LIN {X 0,Y 571.544,Z 581.049,A -85,B 0,C 180,E1 -1504.136,E2 -1504.136} C_VEL
LIN {X 0,Y 571.308,Z 601.407,A -85,B 0,C 180,E1 -1504.632,E2 -1504.632} C_VEL
LIN {X 0,Y 570.995,Z 621.202,A -85,B 0,C 180,E1 -1505.305,E2 -1505.305} C_VEL
LIN {X 0,Y 570.609,Z 639.891,A -85,B 0,C 180,E1 -1506.125,E2 -1506.125} C_VEL
LIN {X 0,Y 570.21,Z 658.766,A -85,B 0,C 180,E1 -1507.147,E2 -1507.147} C_VEL
LIN {X 0,Y 569.785,Z 677.478,A -85,B 0,C 180,E1 -1508.378,E2 -1508.378} C_VEL
LIN {X 0,Y 569.391,Z 694.356,A -85,B 0,C 180,E1 -1509.704,E2 -1509.704} C_VEL
LIN {X 0,Y 569.023,Z 710.417,A -85,B 0,C 180,E1 -1511.191,E2 -1511.191} C_VEL
LIN {X 0,Y 568.698,Z 725.365,A -85,B 0,C 180,E1 -1512.822,E2 -1512.822} C_VEL
LIN {X 0,Y 568.433,Z 739.137,A -85,B 0,C 180,E1 -1514.598,E2 -1514.598} C_VEL
LIN {X 0,Y 568.219,Z 751.298,A -85,B 0,C 180,E1 -1516.467,E2 -1516.467} C_VEL
LIN {X 0,Y 568.077,Z 761.373,A -85,B 0,C 180,E1 -1518.323,E2 -1518.323} C_VEL
LIN {X 0,Y 567.993,Z 770.289,A -85,B 0,C 180,E1 -1520.328,E2 -1520.328} C_VEL
LIN {X 0,Y 567.945,Z 777.475,A -85,B 0,C 180,E1 -1522.372,E2 -1522.372} C_VEL
LIN {X 0,Y 567.92,Z 782.732,A -85,B 0,C 180,E1 -1524.343,E2 -1524.343} C_VEL
LIN {X 0,Y 567.908,Z 786.402,A -85,B 0,C 180,E1 -1526.367,E2 -1526.367} C_VEL
LIN {X 0,Y 567.902,Z 788.441,A -85,B 0,C 180,E1 -1528.387,E2 -1528.387} C_VEL
LIN {X 0,Y 567.9,Z 788.895,A -85,B 0,C 180,E1 -1530.505,E2 -1530.505} C_VEL
LIN {X 0,Y 567.907,Z 787.727,A -85,B 0,C 180,E1 -1532.524,E2 -1532.524} C_VEL
LIN {X 0,Y 567.913,Z 784.97,A -85,B 0,C 180,E1 -1534.545,E2 -1534.545} C_VEL
LIN {X 0,Y 567.931,Z 780.48,A -85,B 0,C 180,E1 -1536.572,E2 -1536.572} C_VEL
LIN {X 0,Y 567.969,Z 774.262,A -85,B 0,C 180,E1 -1538.607,E2 -1538.607} C_VEL
LIN {X 0,Y 568.028,Z 766.175,A -85,B 0,C 180,E1 -1540.652,E2 -1540.652} C_VEL
LIN {X 0,Y 568.143,Z 756.561,A -85,B 0,C 180,E1 -1542.606,E2 -1542.606} C_VEL
LIN {X 0,Y 568.325,Z 745.488,A -85,B 0,C 180,E1 -1544.468,E2 -1544.468} C_VEL
LIN {X 0,Y 568.551,Z 732.933,A -85,B 0,C 180,E1 -1546.238,E2 -1546.238} C_VEL
LIN {X 0,Y 568.832,Z 718.879,A -85,B 0,C 180,E1 -1547.916,E2 -1547.916} C_VEL
LIN {X 0,Y 569.169,Z 703.833,A -85,B 0,C 180,E1 -1549.445,E2 -1549.445} C_VEL
LIN {X 0,Y 569.551,Z 687.283,A -85,B 0,C 180,E1 -1550.878,E2 -1550.878} C_VEL
LIN {X 0,Y 569.976,Z 668.941,A -85,B 0,C 180,E1 -1552.213,E2 -1552.213} C_VEL
LIN {X 0,Y 570.388,Z 650.263,A -85,B 0,C 180,E1 -1553.34,E2 -1553.34} C_VEL
LIN {X 0,Y 570.784,Z 631.791,A -85,B 0,C 180,E1 -1554.255,E2 -1554.255} C_VEL
LIN {X 0,Y 571.16,Z 611.854,A -85,B 0,C 180,E1 -1555.038,E2 -1555.038} C_VEL
LIN {X 0,Y 571.428,Z 591.582,A -85,B 0,C 180,E1 -1555.63,E2 -1555.63} C_VEL
LIN {X 0,Y 571.638,Z 571.154,A -85,B 0,C 180,E1 -1556.037,E2 -1556.037} C_VEL
LIN {X 0,Y 572.618,Z 333.536,A -85,B 0,C 180,E1 -1559.297,E2 -1559.297} C_VEL
LIN {X 0,Y 572.442,Z 320.457,A -85,B 0,C 180,E1 -1559.491,E2 -1559.491} C_VEL
LIN {X 0,Y 571.564,Z 314.836,A -85,B 0,C 180,E1 -1559.646,E2 -1559.646} C_VEL
LIN {X 0,Y 572.165,Z 276.654,A -85,B 0,C 180,E1 -1562.244,E2 -1562.244} C_VEL
LIN {X 0,Y 568.247,Z 266.023,A -85,B 0,C 180,E1 -1563.279,E2 -1563.279} C_VEL
LIN {X 0,Y 568.203,Z 265.709,A -85,B 0,C 180,E1 -1564.149,E2 -1564.149} C_VEL
LIN {X 0,Y 568.186,Z 265.71,A -85,B 0,C 180,E1 -1567.509,E2 -1567.509} C_VEL
LIN {X 0,Y 568.221,Z 265.707,A -85,B 0,C 180,E1 -1570.756,E2 -1570.756} C_VEL
LIN {X 0,Y 568.185,Z 265.706,A -85,B 0,C 180,E1 -1574.036,E2 -1574.036} C_VEL
LIN {X 0,Y 568.192,Z 265.71,A -85,B 0,C 180,E1 -1577.356,E2 -1577.356} C_VEL
LIN {X 0,Y 568.224,Z 265.704,A -85,B 0,C 180,E1 -1580.577,E2 -1580.577} C_VEL
LIN {X 0,Y 568.171,Z 265.709,A -85,B 0,C 180,E1 -1583.752,E2 -1583.752} C_VEL
LIN {X 0,Y 568.219,Z 265.709,A -85,B 0,C 180,E1 -1586.942,E2 -1586.942} C_VEL
LIN {X 0,Y 568.251,Z 265.927,A -85,B 0,C 180,E1 -1589.055,E2 -1589.055} C_VEL
LIN {X 0,Y 571.301,Z 275.947,A -85,B 0,C 180,E1 -1590.08,E2 -1590.08} C_VEL
LIN {X 0,Y 570.614,Z 317.064,A -85,B 0,C 180,E1 -1593.297,E2 -1593.297} C_VEL
LIN {X 0,Y 570.322,Z 342.297,A -85,B 0,C 180,E1 -1595.215,E2 -1595.215} C_VEL
LIN {X 0,Y 571.283,Z 349.569,A -85,B 0,C 180,E1 -1595.372,E2 -1595.372} C_VEL
LIN {X 0,Y 570.541,Z 559.942,A -85,B 0,C 180,E1 -1598.191,E2 -1598.191} C_VEL
LIN {X 0,Y 570.341,Z 579.649,A -85,B 0,C 180,E1 -1598.652,E2 -1598.652} C_VEL
LIN {X 0,Y 570.092,Z 598.197,A -85,B 0,C 180,E1 -1599.278,E2 -1599.278} C_VEL
LIN {X 0,Y 569.786,Z 616.477,A -85,B 0,C 180,E1 -1600.097,E2 -1600.097} C_VEL
LIN {X 0,Y 569.463,Z 634.177,A -85,B 0,C 180,E1 -1601.099,E2 -1601.099} C_VEL
LIN {X 0,Y 569.137,Z 650.753,A -85,B 0,C 180,E1 -1602.254,E2 -1602.254} C_VEL
LIN {X 0,Y 568.827,Z 666.254,A -85,B 0,C 180,E1 -1603.561,E2 -1603.561} C_VEL
LIN {X 0,Y 568.552,Z 680.636,A -85,B 0,C 180,E1 -1605.018,E2 -1605.018} C_VEL
LIN {X 0,Y 568.336,Z 693.477,A -85,B 0,C 180,E1 -1606.572,E2 -1606.572} C_VEL
LIN {X 0,Y 568.164,Z 704.809,A -85,B 0,C 180,E1 -1608.221,E2 -1608.221} C_VEL
LIN {X 0,Y 568.047,Z 714.647,A -85,B 0,C 180,E1 -1609.965,E2 -1609.965} C_VEL
LIN {X 0,Y 567.968,Z 722.967,A -85,B 0,C 180,E1 -1611.802,E2 -1611.802} C_VEL
LIN {X 0,Y 567.933,Z 729.712,A -85,B 0,C 180,E1 -1613.734,E2 -1613.734} C_VEL
LIN {X 0,Y 567.911,Z 734.541,A -85,B 0,C 180,E1 -1615.659,E2 -1615.659} C_VEL
LIN {X 0,Y 567.913,Z 737.572,A -85,B 0,C 180,E1 -1617.579,E2 -1617.579} C_VEL
LIN {X 0,Y 567.908,Z 738.885,A -85,B 0,C 180,E1 -1619.496,E2 -1619.496} C_VEL
LIN {X 0,Y 567.912,Z 738.466,A -85,B 0,C 180,E1 -1621.514,E2 -1621.514} C_VEL
LIN {X 0,Y 567.911,Z 736.336,A -85,B 0,C 180,E1 -1623.432,E2 -1623.432} C_VEL
LIN {X 0,Y 567.922,Z 732.454,A -85,B 0,C 180,E1 -1625.354,E2 -1625.354} C_VEL
LIN {X 0,Y 567.95,Z 726.724,A -85,B 0,C 180,E1 -1627.282,E2 -1627.282} C_VEL
LIN {X 0,Y 568.009,Z 718.999,A -85,B 0,C 180,E1 -1629.218,E2 -1629.218} C_VEL
LIN {X 0,Y 568.11,Z 709.622,A -85,B 0,C 180,E1 -1631.06,E2 -1631.06} C_VEL
LIN {X 0,Y 568.258,Z 698.617,A -85,B 0,C 180,E1 -1632.809,E2 -1632.809} C_VEL
LIN {X 0,Y 568.444,Z 686.814,A -85,B 0,C 180,E1 -1634.36,E2 -1634.36} C_VEL
LIN {X 0,Y 568.684,Z 673.62,A -85,B 0,C 180,E1 -1635.815,E2 -1635.815} C_VEL
LIN {X 0,Y 568.971,Z 658.977,A -85,B 0,C 180,E1 -1637.172,E2 -1637.172} C_VEL
LIN {X 0,Y 569.093,Z 652.545,A -85,B 0,C 180,E1 -1637.695,E2 -1637.695} C_VEL
LIN {X 0,Y 568.272,Z 646.543,A -85,B 0,C 180,E1 -1638.185,E2 -1638.185} C_VEL
LIN {X 0,Y 562.847,Z 631.343,A -85,B 0,C 180,E1 -1639.402,E2 -1639.402} C_VEL
LIN {X 0,Y 562.015,Z 624.834,A -85,B 0,C 180,E1 -1639.822,E2 -1639.822} C_VEL
LIN {X 0,Y 562.403,Z 607.236,A -85,B 0,C 180,E1 -1640.72,E2 -1640.72} C_VEL
LIN {X 0,Y 562.74,Z 588.423,A -85,B 0,C 180,E1 -1641.46,E2 -1641.46} C_VEL
LIN {X 0,Y 563.017,Z 568.721,A -85,B 0,C 180,E1 -1642.021,E2 -1642.021} C_VEL
LIN {X 0,Y 563.199,Z 548.932,A -85,B 0,C 180,E1 -1642.376,E2 -1642.376} C_VEL
LIN {X 0,Y 563.871,Z 348.428,A -85,B 0,C 180,E1 -1645.08,E2 -1645.08} C_VEL
LIN {X 0,Y 562.822,Z 342.045,A -85,B 0,C 180,E1 -1645.237,E2 -1645.237} C_VEL
LIN {X 0,Y 563.583,Z 299.244,A -85,B 0,C 180,E1 -1648.575,E2 -1648.575} C_VEL
LIN {X 0,Y 563.903,Z 277.869,A -85,B 0,C 180,E1 -1650.287,E2 -1650.287} C_VEL
LIN {X 0,Y 560.31,Z 266.962,A -85,B 0,C 180,E1 -1651.432,E2 -1651.432} C_VEL
LIN {X 0,Y 560.233,Z 266.674,A -85,B 0,C 180,E1 -1654.331,E2 -1654.331} C_VEL
LIN {X 0,Y 560.264,Z 266.693,A -85,B 0,C 180,E1 -1657.615,E2 -1657.615} C_VEL
LIN {X 0,Y 560.282,Z 266.696,A -85,B 0,C 180,E1 -1660.915,E2 -1660.915} C_VEL
LIN {X 0,Y 560.255,Z 266.695,A -85,B 0,C 180,E1 -1664.251,E2 -1664.251} C_VEL
LIN {X 0,Y 560.276,Z 266.69,A -85,B 0,C 180,E1 -1667.632,E2 -1667.632} C_VEL
LIN {X 0,Y 560.269,Z 266.695,A -85,B 0,C 180,E1 -1670.952,E2 -1670.952} C_VEL
LIN {X 0,Y 560.273,Z 266.696,A -85,B 0,C 180,E1 -1674.298,E2 -1674.298} C_VEL
LIN {X 0,Y 560.279,Z 266.689,A -85,B 0,C 180,E1 -1677.63,E2 -1677.63} C_VEL
LIN {X 0,Y 560.25,Z 266.692,A -85,B 0,C 180,E1 -1680.985,E2 -1680.985} C_VEL
LIN {X 0,Y 560.279,Z 266.694,A -85,B 0,C 180,E1 -1684.319,E2 -1684.319} C_VEL
LIN {X 0,Y 560.272,Z 266.692,A -85,B 0,C 180,E1 -1687.658,E2 -1687.658} C_VEL
LIN {X 0,Y 560.23,Z 266.696,A -85,B 0,C 180,E1 -1690.936,E2 -1690.936} C_VEL
LIN {X 0,Y 560.275,Z 266.694,A -85,B 0,C 180,E1 -1694.154,E2 -1694.154} C_VEL
LIN {X 0,Y 560.225,Z 266.696,A -85,B 0,C 180,E1 -1697.318,E2 -1697.318} C_VEL
LIN {X 0,Y 560.209,Z 266.692,A -85,B 0,C 180,E1 -1700.652,E2 -1700.652} C_VEL
LIN {X 0,Y 560.309,Z 266.955,A -85,B 0,C 180,E1 -1701.921,E2 -1701.921} C_VEL
LIN {X 0,Y 563.12,Z 276.791,A -85,B 0,C 180,E1 -1702.859,E2 -1702.859} C_VEL
LIN {X 0,Y 563.06,Z 315.928,A -85,B 0,C 180,E1 -1705.875,E2 -1705.875} C_VEL
LIN {X 0,Y 562.759,Z 357.058,A -85,B 0,C 180,E1 -1709.032,E2 -1709.032} C_VEL
LIN {X 0,Y 562.252,Z 395.027,A -85,B 0,C 180,E1 -1711.952,E2 -1711.952} C_VEL
LIN {X 0,Y 561.645,Z 439.417,A -85,B 0,C 180,E1 -1715.362,E2 -1715.362} C_VEL
LIN {X 0,Y 561.272,Z 472.478,A -85,B 0,C 180,E1 -1717.844,E2 -1717.844} C_VEL
LIN {X 0,Y 561.834,Z 480.229,A -85,B 0,C 180,E1 -1717.975,E2 -1717.975} C_VEL
LIN {X 0,Y 561.421,Z 615.352,A -85,B 0,C 180,E1 -1719.752,E2 -1719.752} C_VEL
LIN {X 0,Y 561.296,Z 631.802,A -85,B 0,C 180,E1 -1720.167,E2 -1720.167} C_VEL
LIN {X 0,Y 561.1,Z 648.005,A -85,B 0,C 180,E1 -1720.783,E2 -1720.783} C_VEL
LIN {X 0,Y 560.866,Z 663.048,A -85,B 0,C 180,E1 -1721.568,E2 -1721.568} C_VEL
LIN {X 0,Y 560.64,Z 677.243,A -85,B 0,C 180,E1 -1722.524,E2 -1722.524} C_VEL
LIN {X 0,Y 560.42,Z 690.634,A -85,B 0,C 180,E1 -1723.673,E2 -1723.673} C_VEL
LIN {X 0,Y 560.245,Z 702.045,A -85,B 0,C 180,E1 -1724.89,E2 -1724.89} C_VEL
LIN {X 0,Y 560.103,Z 712.396,A -85,B 0,C 180,E1 -1726.275,E2 -1726.275} C_VEL
LIN {X 0,Y 560.008,Z 721.264,A -85,B 0,C 180,E1 -1727.775,E2 -1727.775} C_VEL
LIN {X 0,Y 559.948,Z 728.518,A -85,B 0,C 180,E1 -1729.396,E2 -1729.396} C_VEL
LIN {X 0,Y 559.928,Z 733.575,A -85,B 0,C 180,E1 -1730.945,E2 -1730.945} C_VEL
LIN {X 0,Y 559.916,Z 737.056,A -85,B 0,C 180,E1 -1732.597,E2 -1732.597} C_VEL
LIN {X 0,Y 559.918,Z 738.783,A -85,B 0,C 180,E1 -1734.248,E2 -1734.248} C_VEL
LIN {X 0,Y 559.915,Z 738.784,A -85,B 0,C 180,E1 -1735.839,E2 -1735.839} C_VEL
LIN {X 0,Y 559.916,Z 736.969,A -85,B 0,C 180,E1 -1737.547,E2 -1737.547} C_VEL
LIN {X 0,Y 559.929,Z 733.494,A -85,B 0,C 180,E1 -1739.174,E2 -1739.174} C_VEL
LIN {X 0,Y 559.953,Z 728.002,A -85,B 0,C 180,E1 -1740.827,E2 -1740.827} C_VEL
LIN {X 0,Y 560.011,Z 720.905,A -85,B 0,C 180,E1 -1742.385,E2 -1742.385} C_VEL
LIN {X 0,Y 560.11,Z 711.882,A -85,B 0,C 180,E1 -1743.892,E2 -1743.892} C_VEL
LIN {X 0,Y 560.245,Z 702.046,A -85,B 0,C 180,E1 -1745.199,E2 -1745.199} C_VEL
LIN {X 0,Y 560.425,Z 690.324,A -85,B 0,C 180,E1 -1746.447,E2 -1746.447} C_VEL
LIN {X 0,Y 560.644,Z 677.033,A -85,B 0,C 180,E1 -1747.582,E2 -1747.582} C_VEL
LIN {X 0,Y 560.868,Z 662.899,A -85,B 0,C 180,E1 -1748.531,E2 -1748.531} C_VEL
LIN {X 0,Y 561.089,Z 648.335,A -85,B 0,C 180,E1 -1749.292,E2 -1749.292} C_VEL
LIN {X 0,Y 561.289,Z 632.212,A -85,B 0,C 180,E1 -1749.91,E2 -1749.91} C_VEL
LIN {X 0,Y 561.405,Z 615.816,A -85,B 0,C 180,E1 -1750.33,E2 -1750.33} C_VEL
LIN {X 0,Y 561.631,Z 540.614,A -85,B 0,C 180,E1 -1751.332,E2 -1751.332} C_VEL
LIN {X 0,Y 561.621,Z 475.594,A -85,B 0,C 180,E1 -1752.183,E2 -1752.183} C_VEL
LIN {X 0,Y 561.244,Z 472.411,A -85,B 0,C 180,E1 -1752.249,E2 -1752.249} C_VEL
LIN {X 0,Y 561.705,Z 433.531,A -85,B 0,C 180,E1 -1755.178,E2 -1755.178} C_VEL
LIN {X 0,Y 562.301,Z 390.839,A -85,B 0,C 180,E1 -1758.467,E2 -1758.467} C_VEL
LIN {X 0,Y 562.735,Z 360.838,A -85,B 0,C 180,E1 -1760.773,E2 -1760.773} C_VEL
LIN {X 0,Y 562.922,Z 318.216,A -85,B 0,C 180,E1 -1763.99,E2 -1763.99} C_VEL
LIN {X 0,Y 562.881,Z 280.091,A -85,B 0,C 180,E1 -1766.891,E2 -1766.891} C_VEL
LIN {X 0,Y 562.592,Z 274.842,A -85,B 0,C 180,E1 -1767.297,E2 -1767.297} C_VEL
LIN {X 0,Y 560.307,Z 267.002,A -85,B 0,C 180,E1 -1768.025,E2 -1768.025} C_VEL
LIN {X 0,Y 560.264,Z 266.699,A -85,B 0,C 180,E1 -1768.832,E2 -1768.832} C_VEL
LIN {X 0,Y 560.268,Z 266.7,A -85,B 0,C 180,E1 -1772.123,E2 -1772.123} C_VEL
LIN {X 0,Y 560.234,Z 266.697,A -85,B 0,C 180,E1 -1775.427,E2 -1775.427} C_VEL
LIN {X 0,Y 560.282,Z 266.692,A -85,B 0,C 180,E1 -1778.671,E2 -1778.671} C_VEL
LIN {X 0,Y 560.246,Z 266.695,A -85,B 0,C 180,E1 -1781.908,E2 -1781.908} C_VEL
LIN {X 0,Y 560.241,Z 266.693,A -85,B 0,C 180,E1 -1785.319,E2 -1785.319} C_VEL
LIN {X 0,Y 560.282,Z 266.695,A -85,B 0,C 180,E1 -1788.575,E2 -1788.575} C_VEL
LIN {X 0,Y 560.238,Z 266.695,A -85,B 0,C 180,E1 -1791.791,E2 -1791.791} C_VEL
LIN {X 0,Y 560.268,Z 266.691,A -85,B 0,C 180,E1 -1795.086,E2 -1795.086} C_VEL
LIN {X 0,Y 560.272,Z 266.698,A -85,B 0,C 180,E1 -1798.363,E2 -1798.363} C_VEL
LIN {X 0,Y 560.24,Z 266.693,A -85,B 0,C 180,E1 -1801.636,E2 -1801.636} C_VEL
LIN {X 0,Y 560.283,Z 266.692,A -85,B 0,C 180,E1 -1804.914,E2 -1804.914} C_VEL
LIN {X 0,Y 560.251,Z 266.697,A -85,B 0,C 180,E1 -1808.208,E2 -1808.208} C_VEL
LIN {X 0,Y 560.248,Z 266.692,A -85,B 0,C 180,E1 -1811.55,E2 -1811.55} C_VEL
LIN {X 0,Y 560.281,Z 266.694,A -85,B 0,C 180,E1 -1814.785,E2 -1814.785} C_VEL
LIN {X 0,Y 560.245,Z 266.695,A -85,B 0,C 180,E1 -1818.091,E2 -1818.091} C_VEL
LIN {X 0,Y 560.262,Z 266.69,A -85,B 0,C 180,E1 -1821.459,E2 -1821.459} C_VEL
LIN {X 0,Y 560.283,Z 266.697,A -85,B 0,C 180,E1 -1824.795,E2 -1824.795} C_VEL
LIN {X 0,Y 560.244,Z 266.694,A -85,B 0,C 180,E1 -1828.109,E2 -1828.109} C_VEL
LIN {X 0,Y 560.272,Z 266.69,A -85,B 0,C 180,E1 -1831.46,E2 -1831.46} C_VEL
LIN {X 0,Y 560.278,Z 266.698,A -85,B 0,C 180,E1 -1834.828,E2 -1834.828} C_VEL
LIN {X 0,Y 560.245,Z 266.694,A -85,B 0,C 180,E1 -1838.133,E2 -1838.133} C_VEL
LIN {X 0,Y 560.28,Z 266.691,A -85,B 0,C 180,E1 -1841.458,E2 -1841.458} C_VEL
LIN {X 0,Y 560.278,Z 266.698,A -85,B 0,C 180,E1 -1844.822,E2 -1844.822} C_VEL
LIN {X 0,Y 560.247,Z 266.695,A -85,B 0,C 180,E1 -1848.13,E2 -1848.13} C_VEL
LIN {X 0,Y 560.282,Z 266.694,A -85,B 0,C 180,E1 -1851.41,E2 -1851.41} C_VEL
LIN {X 0,Y 560.268,Z 266.669,A -85,B 0,C 180,E1 -1854.802,E2 -1854.802} C_VEL
LIN {X 0,Y 560.278,Z 266.906,A -85,B 0,C 180,E1 -1856.229,E2 -1856.229} C_VEL
LIN {X 0,Y 561.758,Z 271.085,A -85,B 0,C 180,E1 -1856.683,E2 -1856.683} C_VEL
LIN {X 0,Y 565.073,Z 279.818,A -85,B 0,C 180,E1 -1857.527,E2 -1857.527} C_VEL
LIN {X 0,Y 564.444,Z 315.729,A -85,B 0,C 180,E1 -1859.977,E2 -1859.977} C_VEL
LIN {X 0,Y 565.686,Z 324.502,A -85,B 0,C 180,E1 -1860.179,E2 -1860.179} C_VEL
LIN {X 0,Y 564.555,Z 553.958,A -85,B 0,C 180,E1 -1863.36,E2 -1863.36} C_VEL
LIN {X 0,Y 564.325,Z 581.698,A -85,B 0,C 180,E1 -1863.795,E2 -1863.795} C_VEL
LIN {X 0,Y 564.036,Z 601.947,A -85,B 0,C 180,E1 -1864.299,E2 -1864.299} C_VEL
LIN {X 0,Y 563.663,Z 621.652,A -85,B 0,C 180,E1 -1864.979,E2 -1864.979} C_VEL
LIN {X 0,Y 563.193,Z 640.59,A -85,B 0,C 180,E1 -1865.825,E2 -1865.825} C_VEL
LIN {X 0,Y 562.703,Z 659.659,A -85,B 0,C 180,E1 -1866.879,E2 -1866.879} C_VEL
LIN {X 0,Y 562.187,Z 678.21,A -85,B 0,C 180,E1 -1868.126,E2 -1868.126} C_VEL
LIN {X 0,Y 561.687,Z 695.631,A -85,B 0,C 180,E1 -1869.527,E2 -1869.527} C_VEL
LIN {X 0,Y 561.246,Z 711.43,A -85,B 0,C 180,E1 -1871.028,E2 -1871.028} C_VEL
LIN {X 0,Y 560.855,Z 726.217,A -85,B 0,C 180,E1 -1872.681,E2 -1872.681} C_VEL
LIN {X 0,Y 560.539,Z 739.871,A -85,B 0,C 180,E1 -1874.482,E2 -1874.482} C_VEL
LIN {X 0,Y 560.285,Z 751.932,A -85,B 0,C 180,E1 -1876.377,E2 -1876.377} C_VEL
LIN {X 0,Y 560.111,Z 762.401,A -85,B 0,C 180,E1 -1878.364,E2 -1878.364} C_VEL
LIN {X 0,Y 560.008,Z 770.879,A -85,B 0,C 180,E1 -1880.34,E2 -1880.34} C_VEL
LIN {X 0,Y 559.947,Z 777.903,A -85,B 0,C 180,E1 -1882.408,E2 -1882.408} C_VEL
LIN {X 0,Y 559.916,Z 783.145,A -85,B 0,C 180,E1 -1884.468,E2 -1884.468} C_VEL
LIN {X 0,Y 559.903,Z 786.711,A -85,B 0,C 180,E1 -1886.52,E2 -1886.52} C_VEL
LIN {X 0,Y 559.9,Z 788.575,A -85,B 0,C 180,E1 -1888.569,E2 -1888.569} C_VEL
LIN {X 0,Y 559.901,Z 788.873,A -85,B 0,C 180,E1 -1890.615,E2 -1890.615} C_VEL
LIN {X 0,Y 559.911,Z 787.504,A -85,B 0,C 180,E1 -1892.765,E2 -1892.765} C_VEL
LIN {X 0,Y 559.92,Z 784.519,A -85,B 0,C 180,E1 -1894.845,E2 -1894.845} C_VEL
LIN {X 0,Y 559.936,Z 779.972,A -85,B 0,C 180,E1 -1896.872,E2 -1896.872} C_VEL
LIN {X 0,Y 559.976,Z 773.909,A -85,B 0,C 180,E1 -1898.834,E2 -1898.834} C_VEL
LIN {X 0,Y 560.054,Z 766.176,A -85,B 0,C 180,E1 -1900.805,E2 -1900.805} C_VEL
LIN {X 0,Y 560.192,Z 757.134,A -85,B 0,C 180,E1 -1902.683,E2 -1902.683} C_VEL
LIN {X 0,Y 560.409,Z 746.174,A -85,B 0,C 180,E1 -1904.571,E2 -1904.571} C_VEL
LIN {X 0,Y 560.68,Z 733.606,A -85,B 0,C 180,E1 -1906.381,E2 -1906.381} C_VEL
LIN {X 0,Y 561.017,Z 719.806,A -85,B 0,C 180,E1 -1908.067,E2 -1908.067} C_VEL
LIN {X 0,Y 561.417,Z 705.224,A -85,B 0,C 180,E1 -1909.589,E2 -1909.589} C_VEL
LIN {X 0,Y 561.906,Z 687.948,A -85,B 0,C 180,E1 -1911.121,E2 -1911.121} C_VEL
LIN {X 0,Y 562.422,Z 669.746,A -85,B 0,C 180,E1 -1912.472,E2 -1912.472} C_VEL
LIN {X 0,Y 562.917,Z 651.36,A -85,B 0,C 180,E1 -1913.607,E2 -1913.607} C_VEL
LIN {X 0,Y 563.397,Z 633.055,A -85,B 0,C 180,E1 -1914.538,E2 -1914.538} C_VEL
LIN {X 0,Y 563.826,Z 613.331,A -85,B 0,C 180,E1 -1915.33,E2 -1915.33} C_VEL
LIN {X 0,Y 564.155,Z 593.353,A -85,B 0,C 180,E1 -1915.937,E2 -1915.937} C_VEL
LIN {X 0,Y 564.441,Z 572.22,A -85,B 0,C 180,E1 -1916.377,E2 -1916.377} C_VEL
LIN {X 0,Y 565.636,Z 334.299,A -85,B 0,C 180,E1 -1919.684,E2 -1919.684} C_VEL
LIN {X 0,Y 565.47,Z 321.725,A -85,B 0,C 180,E1 -1919.873,E2 -1919.873} C_VEL
LIN {X 0,Y 564.376,Z 315.078,A -85,B 0,C 180,E1 -1920.047,E2 -1920.047} C_VEL
LIN {X 0,Y 565.074,Z 279.781,A -85,B 0,C 180,E1 -1922.476,E2 -1922.476} C_VEL
LIN {X 0,Y 560.299,Z 267.044,A -85,B 0,C 180,E1 -1923.739,E2 -1923.739} C_VEL
LIN {X 0,Y 560.281,Z 266.696,A -85,B 0,C 180,E1 -1924.466,E2 -1924.466} C_VEL
LIN {X 0,Y 560.243,Z 266.698,A -85,B 0,C 180,E1 -1927.757,E2 -1927.757} C_VEL
LIN {X 0,Y 560.28,Z 266.699,A -85,B 0,C 180,E1 -1931.051,E2 -1931.051} C_VEL
LIN {X 0,Y 560.273,Z 266.693,A -85,B 0,C 180,E1 -1934.393,E2 -1934.393} C_VEL
LIN {X 0,Y 560.238,Z 266.697,A -85,B 0,C 180,E1 -1937.714,E2 -1937.714} C_VEL
LIN {X 0,Y 560.285,Z 266.697,A -85,B 0,C 180,E1 -1940.954,E2 -1940.954} C_VEL
LIN {X 0,Y 560.242,Z 266.697,A -85,B 0,C 180,E1 -1944.171,E2 -1944.171} C_VEL
LIN {X 0,Y 560.235,Z 266.702,A -85,B 0,C 180,E1 -1947.584,E2 -1947.584} C_VEL
LIN {X 0,Y 560.316,Z 266.965,A -85,B 0,C 180,E1 -1948.657,E2 -1948.657} C_VEL
LIN {X 0,Y 563.994,Z 278.837,A -85,B 0,C 180,E1 -1949.887,E2 -1949.887} C_VEL
LIN {X 0,Y 563.168,Z 320.602,A -85,B 0,C 180,E1 -1953.195,E2 -1953.195} C_VEL
LIN {X 0,Y 562.846,Z 342.314,A -85,B 0,C 180,E1 -1954.863,E2 -1954.863} C_VEL
LIN {X 0,Y 564.008,Z 350.714,A -85,B 0,C 180,E1 -1955.048,E2 -1955.048} C_VEL
LIN {X 0,Y 563.116,Z 559.798,A -85,B 0,C 180,E1 -1957.885,E2 -1957.885} C_VEL
LIN {X 0,Y 562.874,Z 579.546,A -85,B 0,C 180,E1 -1958.351,E2 -1958.351} C_VEL
LIN {X 0,Y 562.57,Z 598.215,A -85,B 0,C 180,E1 -1958.988,E2 -1958.988} C_VEL
LIN {X 0,Y 562.198,Z 616.486,A -85,B 0,C 180,E1 -1959.817,E2 -1959.817} C_VEL
LIN {X 0,Y 561.806,Z 634.182,A -85,B 0,C 180,E1 -1960.831,E2 -1960.831} C_VEL
LIN {X 0,Y 561.413,Z 650.716,A -85,B 0,C 180,E1 -1961.998,E2 -1961.998} C_VEL
LIN {X 0,Y 561.036,Z 666.26,A -85,B 0,C 180,E1 -1963.326,E2 -1963.326} C_VEL
LIN {X 0,Y 560.702,Z 680.641,A -85,B 0,C 180,E1 -1964.804,E2 -1964.804} C_VEL
LIN {X 0,Y 560.439,Z 693.485,A -85,B 0,C 180,E1 -1966.379,E2 -1966.379} C_VEL
LIN {X 0,Y 560.226,Z 704.816,A -85,B 0,C 180,E1 -1968.052,E2 -1968.052} C_VEL
LIN {X 0,Y 560.085,Z 714.653,A -85,B 0,C 180,E1 -1969.821,E2 -1969.821} C_VEL
LIN {X 0,Y 559.984,Z 722.97,A -85,B 0,C 180,E1 -1971.685,E2 -1971.685} C_VEL
LIN {X 0,Y 559.938,Z 729.715,A -85,B 0,C 180,E1 -1973.644,E2 -1973.644} C_VEL
LIN {X 0,Y 559.912,Z 734.545,A -85,B 0,C 180,E1 -1975.596,E2 -1975.596} C_VEL
LIN {X 0,Y 559.913,Z 737.575,A -85,B 0,C 180,E1 -1977.544,E2 -1977.544} C_VEL
LIN {X 0,Y 559.908,Z 738.885,A -85,B 0,C 180,E1 -1979.489,E2 -1979.489} C_VEL
LIN {X 0,Y 559.912,Z 738.467,A -85,B 0,C 180,E1 -1981.535,E2 -1981.535} C_VEL
LIN {X 0,Y 559.91,Z 736.338,A -85,B 0,C 180,E1 -1983.481,E2 -1983.481} C_VEL
LIN {X 0,Y 559.924,Z 732.455,A -85,B 0,C 180,E1 -1985.431,E2 -1985.431} C_VEL
LIN {X 0,Y 559.957,Z 726.723,A -85,B 0,C 180,E1 -1987.387,E2 -1987.387} C_VEL
LIN {X 0,Y 560.036,Z 718.997,A -85,B 0,C 180,E1 -1989.351,E2 -1989.351} C_VEL
LIN {X 0,Y 560.157,Z 709.621,A -85,B 0,C 180,E1 -1991.219,E2 -1991.219} C_VEL
LIN {X 0,Y 560.34,Z 698.616,A -85,B 0,C 180,E1 -1992.993,E2 -1992.993} C_VEL
LIN {X 0,Y 560.569,Z 686.811,A -85,B 0,C 180,E1 -1994.566,E2 -1994.566} C_VEL
LIN {X 0,Y 560.869,Z 673.245,A -85,B 0,C 180,E1 -1996.079,E2 -1996.079} C_VEL
LIN {X 0,Y 561.22,Z 658.578,A -85,B 0,C 180,E1 -1997.451,E2 -1997.451} C_VEL
LIN {X 0,Y 561.616,Z 642.337,A -85,B 0,C 180,E1 -1998.713,E2 -1998.713} C_VEL
LIN {X 0,Y 562.015,Z 624.834,A -85,B 0,C 180,E1 -1999.822,E2 -1999.822} C_VEL
LIN {X 0,Y 561.226,Z 618.186,A -85,B 0,C 180,E1 -2000.225,E2 -2000.225} C_VEL
LIN {X 0,Y 555.927,Z 601.44,A -85,B 0,C 180,E1 -2001.23,E2 -2001.23} C_VEL
LIN {X 0,Y 555.124,Z 594.384,A -85,B 0,C 180,E1 -2001.548,E2 -2001.548} C_VEL
LIN {X 0,Y 555.482,Z 575.161,A -85,B 0,C 180,E1 -2002.168,E2 -2002.168} C_VEL
LIN {X 0,Y 555.742,Z 555.75,A -85,B 0,C 180,E1 -2002.586,E2 -2002.586} C_VEL
LIN {X 0,Y 556.621,Z 349.619,A -85,B 0,C 180,E1 -2005.412,E2 -2005.412} C_VEL
LIN {X 0,Y 555.366,Z 342.045,A -85,B 0,C 180,E1 -2005.601,E2 -2005.601} C_VEL
LIN {X 0,Y 556.271,Z 299.379,A -85,B 0,C 180,E1 -2008.974,E2 -2008.974} C_VEL
LIN {X 0,Y 556.522,Z 280.46,A -85,B 0,C 180,E1 -2010.516,E2 -2010.516} C_VEL
LIN {X 0,Y 552.328,Z 267.902,A -85,B 0,C 180,E1 -2011.868,E2 -2011.868} C_VEL
LIN {X 0,Y 552.336,Z 267.663,A -85,B 0,C 180,E1 -2014.911,E2 -2014.911} C_VEL
LIN {X 0,Y 552.305,Z 267.685,A -85,B 0,C 180,E1 -2018.254,E2 -2018.254} C_VEL
LIN {X 0,Y 552.329,Z 267.679,A -85,B 0,C 180,E1 -2021.634,E2 -2021.634} C_VEL
LIN {X 0,Y 552.339,Z 267.686,A -85,B 0,C 180,E1 -2024.943,E2 -2024.943} C_VEL
LIN {X 0,Y 552.324,Z 267.684,A -85,B 0,C 180,E1 -2028.232,E2 -2028.232} C_VEL
LIN {X 0,Y 552.343,Z 267.678,A -85,B 0,C 180,E1 -2031.617,E2 -2031.617} C_VEL
LIN {X 0,Y 552.324,Z 267.683,A -85,B 0,C 180,E1 -2034.98,E2 -2034.98} C_VEL
LIN {X 0,Y 552.341,Z 267.686,A -85,B 0,C 180,E1 -2038.333,E2 -2038.333} C_VEL
LIN {X 0,Y 552.342,Z 267.677,A -85,B 0,C 180,E1 -2041.687,E2 -2041.687} C_VEL
LIN {X 0,Y 552.304,Z 267.68,A -85,B 0,C 180,E1 -2045.05,E2 -2045.05} C_VEL
LIN {X 0,Y 552.333,Z 267.683,A -85,B 0,C 180,E1 -2048.327,E2 -2048.327} C_VEL
LIN {X 0,Y 552.325,Z 267.683,A -85,B 0,C 180,E1 -2051.639,E2 -2051.639} C_VEL
LIN {X 0,Y 552.28,Z 267.68,A -85,B 0,C 180,E1 -2054.887,E2 -2054.887} C_VEL
LIN {X 0,Y 552.331,Z 267.688,A -85,B 0,C 180,E1 -2058.089,E2 -2058.089} C_VEL
LIN {X 0,Y 552.275,Z 267.688,A -85,B 0,C 180,E1 -2061.305,E2 -2061.305} C_VEL
LIN {X 0,Y 552.348,Z 268.019,A -85,B 0,C 180,E1 -2061.594,E2 -2061.594} C_VEL
LIN {X 0,Y 555.682,Z 279.748,A -85,B 0,C 180,E1 -2062.711,E2 -2062.711} C_VEL
LIN {X 0,Y 555.546,Z 319.159,A -85,B 0,C 180,E1 -2065.767,E2 -2065.767} C_VEL
LIN {X 0,Y 555.163,Z 359.793,A -85,B 0,C 180,E1 -2068.915,E2 -2068.915} C_VEL
LIN {X 0,Y 554.627,Z 395.794,A -85,B 0,C 180,E1 -2071.703,E2 -2071.703} C_VEL
LIN {X 0,Y 553.969,Z 440.023,A -85,B 0,C 180,E1 -2075.125,E2 -2075.125} C_VEL
LIN {X 0,Y 553.523,Z 472.352,A -85,B 0,C 180,E1 -2077.589,E2 -2077.589} C_VEL
LIN {X 0,Y 554.186,Z 480.588,A -85,B 0,C 180,E1 -2077.736,E2 -2077.736} C_VEL
LIN {X 0,Y 553.701,Z 615.423,A -85,B 0,C 180,E1 -2079.535,E2 -2079.535} C_VEL
LIN {X 0,Y 553.549,Z 631.717,A -85,B 0,C 180,E1 -2079.952,E2 -2079.952} C_VEL
LIN {X 0,Y 553.324,Z 647.903,A -85,B 0,C 180,E1 -2080.573,E2 -2080.573} C_VEL
LIN {X 0,Y 553.052,Z 662.877,A -85,B 0,C 180,E1 -2081.364,E2 -2081.364} C_VEL
LIN {X 0,Y 552.78,Z 676.977,A -85,B 0,C 180,E1 -2082.322,E2 -2082.322} C_VEL
LIN {X 0,Y 552.532,Z 689.984,A -85,B 0,C 180,E1 -2083.445,E2 -2083.445} C_VEL
LIN {X 0,Y 552.317,Z 701.515,A -85,B 0,C 180,E1 -2084.68,E2 -2084.68} C_VEL
LIN {X 0,Y 552.148,Z 711.975,A -85,B 0,C 180,E1 -2086.083,E2 -2086.083} C_VEL
LIN {X 0,Y 552.028,Z 720.937,A -85,B 0,C 180,E1 -2087.605,E2 -2087.605} C_VEL
LIN {X 0,Y 551.961,Z 727.845,A -85,B 0,C 180,E1 -2089.138,E2 -2089.138} C_VEL
LIN {X 0,Y 551.93,Z 733.356,A -85,B 0,C 180,E1 -2090.808,E2 -2090.808} C_VEL
LIN {X 0,Y 551.919,Z 736.92,A -85,B 0,C 180,E1 -2092.471,E2 -2092.471} C_VEL
LIN {X 0,Y 551.918,Z 738.738,A -85,B 0,C 180,E1 -2094.167,E2 -2094.167} C_VEL
LIN {X 0,Y 551.914,Z 738.822,A -85,B 0,C 180,E1 -2095.791,E2 -2095.791} C_VEL
LIN {X 0,Y 551.916,Z 737.077,A -85,B 0,C 180,E1 -2097.512,E2 -2097.512} C_VEL
LIN {X 0,Y 551.93,Z 733.669,A -85,B 0,C 180,E1 -2099.169,E2 -2099.169} C_VEL
LIN {X 0,Y 551.959,Z 728.277,A -85,B 0,C 180,E1 -2100.839,E2 -2100.839} C_VEL
LIN {X 0,Y 552.027,Z 721.222,A -85,B 0,C 180,E1 -2102.429,E2 -2102.429} C_VEL
LIN {X 0,Y 552.143,Z 712.252,A -85,B 0,C 180,E1 -2103.964,E2 -2103.964} C_VEL
LIN {X 0,Y 552.308,Z 702.136,A -85,B 0,C 180,E1 -2105.336,E2 -2105.336} C_VEL
LIN {X 0,Y 552.525,Z 690.435,A -85,B 0,C 180,E1 -2106.601,E2 -2106.601} C_VEL
LIN {X 0,Y 552.765,Z 678.003,A -85,B 0,C 180,E1 -2107.688,E2 -2107.688} C_VEL
LIN {X 0,Y 553.024,Z 664.254,A -85,B 0,C 180,E1 -2108.642,E2 -2108.642} C_VEL
LIN {X 0,Y 553.293,Z 649.215,A -85,B 0,C 180,E1 -2109.456,E2 -2109.456} C_VEL
LIN {X 0,Y 553.53,Z 633.394,A -85,B 0,C 180,E1 -2110.083,E2 -2110.083} C_VEL
LIN {X 0,Y 553.679,Z 617.007,A -85,B 0,C 180,E1 -2110.524,E2 -2110.524} C_VEL
LIN {X 0,Y 553.797,Z 584.698,A -85,B 0,C 180,E1 -2110.986,E2 -2110.986} C_VEL
LIN {X 0,Y 553.976,Z 476.401,A -85,B 0,C 180,E1 -2112.416,E2 -2112.416} C_VEL
LIN {X 0,Y 553.484,Z 472.041,A -85,B 0,C 180,E1 -2112.519,E2 -2112.519} C_VEL
LIN {X 0,Y 554.149,Z 429.88,A -85,B 0,C 180,E1 -2115.748,E2 -2115.748} C_VEL
LIN {X 0,Y 554.787,Z 388.2,A -85,B 0,C 180,E1 -2119.003,E2 -2119.003} C_VEL
LIN {X 0,Y 555.175,Z 355.136,A -85,B 0,C 180,E1 -2121.52,E2 -2121.52} C_VEL
LIN {X 0,Y 555.428,Z 312.632,A -85,B 0,C 180,E1 -2124.769,E2 -2124.769} C_VEL
LIN {X 0,Y 555.275,Z 277.84,A -85,B 0,C 180,E1 -2127.425,E2 -2127.425} C_VEL
LIN {X 0,Y 552.382,Z 267.955,A -85,B 0,C 180,E1 -2128.352,E2 -2128.352} C_VEL
LIN {X 0,Y 552.345,Z 267.684,A -85,B 0,C 180,E1 -2130.537,E2 -2130.537} C_VEL
LIN {X 0,Y 552.309,Z 267.688,A -85,B 0,C 180,E1 -2133.882,E2 -2133.882} C_VEL
LIN {X 0,Y 552.303,Z 267.684,A -85,B 0,C 180,E1 -2137.206,E2 -2137.206} C_VEL
LIN {X 0,Y 552.343,Z 267.684,A -85,B 0,C 180,E1 -2140.434,E2 -2140.434} C_VEL
LIN {X 0,Y 552.297,Z 267.686,A -85,B 0,C 180,E1 -2143.703,E2 -2143.703} C_VEL
LIN {X 0,Y 552.324,Z 267.681,A -85,B 0,C 180,E1 -2147.028,E2 -2147.028} C_VEL
LIN {X 0,Y 552.334,Z 267.688,A -85,B 0,C 180,E1 -2150.308,E2 -2150.308} C_VEL
LIN {X 0,Y 552.299,Z 267.683,A -85,B 0,C 180,E1 -2153.644,E2 -2153.644} C_VEL
LIN {X 0,Y 552.337,Z 267.681,A -85,B 0,C 180,E1 -2156.99,E2 -2156.99} C_VEL
LIN {X 0,Y 552.329,Z 267.687,A -85,B 0,C 180,E1 -2160.311,E2 -2160.311} C_VEL
LIN {X 0,Y 552.302,Z 267.682,A -85,B 0,C 180,E1 -2163.632,E2 -2163.632} C_VEL
LIN {X 0,Y 552.343,Z 267.68,A -85,B 0,C 180,E1 -2166.966,E2 -2166.966} C_VEL
LIN {X 0,Y 552.321,Z 267.685,A -85,B 0,C 180,E1 -2170.324,E2 -2170.324} C_VEL
LIN {X 0,Y 552.304,Z 267.682,A -85,B 0,C 180,E1 -2173.718,E2 -2173.718} C_VEL
LIN {X 0,Y 552.342,Z 267.682,A -85,B 0,C 180,E1 -2176.944,E2 -2176.944} C_VEL
LIN {X 0,Y 552.311,Z 267.685,A -85,B 0,C 180,E1 -2180.229,E2 -2180.229} C_VEL
LIN {X 0,Y 552.31,Z 267.682,A -85,B 0,C 180,E1 -2183.696,E2 -2183.696} C_VEL
LIN {X 0,Y 552.342,Z 267.682,A -85,B 0,C 180,E1 -2187.024,E2 -2187.024} C_VEL
LIN {X 0,Y 552.312,Z 267.684,A -85,B 0,C 180,E1 -2190.336,E2 -2190.336} C_VEL
LIN {X 0,Y 552.312,Z 267.681,A -85,B 0,C 180,E1 -2193.808,E2 -2193.808} C_VEL
LIN {X 0,Y 552.342,Z 267.683,A -85,B 0,C 180,E1 -2197.071,E2 -2197.071} C_VEL
LIN {X 0,Y 552.313,Z 267.685,A -85,B 0,C 180,E1 -2200.398,E2 -2200.398} C_VEL
LIN {X 0,Y 552.323,Z 267.682,A -85,B 0,C 180,E1 -2203.758,E2 -2203.758} C_VEL
LIN {X 0,Y 552.341,Z 267.685,A -85,B 0,C 180,E1 -2207.108,E2 -2207.108} C_VEL
LIN {X 0,Y 552.31,Z 267.686,A -85,B 0,C 180,E1 -2210.416,E2 -2210.416} C_VEL
LIN {X 0,Y 552.321,Z 267.656,A -85,B 0,C 180,E1 -2213.834,E2 -2213.834} C_VEL
LIN {X 0,Y 552.36,Z 267.887,A -85,B 0,C 180,E1 -2215.773,E2 -2215.773} C_VEL
LIN {X 0,Y 554.065,Z 272.818,A -85,B 0,C 180,E1 -2216.296,E2 -2216.296} C_VEL
LIN {X 0,Y 557.956,Z 283.115,A -85,B 0,C 180,E1 -2217.299,E2 -2217.299} C_VEL
LIN {X 0,Y 557.276,Z 315.739,A -85,B 0,C 180,E1 -2219.55,E2 -2219.55} C_VEL
LIN {X 0,Y 558.737,Z 325.763,A -85,B 0,C 180,E1 -2219.788,E2 -2219.788} C_VEL
LIN {X 0,Y 557.399,Z 554.976,A -85,B 0,C 180,E1 -2223.005,E2 -2223.005} C_VEL
LIN {X 0,Y 557.13,Z 582.184,A -85,B 0,C 180,E1 -2223.441,E2 -2223.441} C_VEL
LIN {X 0,Y 556.781,Z 602.596,A -85,B 0,C 180,E1 -2223.961,E2 -2223.961} C_VEL
LIN {X 0,Y 556.348,Z 622.128,A -85,B 0,C 180,E1 -2224.646,E2 -2224.646} C_VEL
LIN {X 0,Y 555.779,Z 641.891,A -85,B 0,C 180,E1 -2225.547,E2 -2225.547} C_VEL
LIN {X 0,Y 555.201,Z 660.724,A -85,B 0,C 180,E1 -2226.615,E2 -2226.615} C_VEL
LIN {X 0,Y 554.601,Z 678.942,A -85,B 0,C 180,E1 -2227.866,E2 -2227.866} C_VEL
LIN {X 0,Y 554.011,Z 696.238,A -85,B 0,C 180,E1 -2229.286,E2 -2229.286} C_VEL
LIN {X 0,Y 553.49,Z 711.936,A -85,B 0,C 180,E1 -2230.807,E2 -2230.807} C_VEL
LIN {X 0,Y 553.04,Z 726.218,A -85,B 0,C 180,E1 -2232.428,E2 -2232.428} C_VEL
LIN {X 0,Y 552.662,Z 739.872,A -85,B 0,C 180,E1 -2234.255,E2 -2234.255} C_VEL
LIN {X 0,Y 552.363,Z 751.931,A -85,B 0,C 180,E1 -2236.177,E2 -2236.177} C_VEL
LIN {X 0,Y 552.149,Z 762.4,A -85,B 0,C 180,E1 -2238.194,E2 -2238.194} C_VEL
LIN {X 0,Y 552.03,Z 770.879,A -85,B 0,C 180,E1 -2240.199,E2 -2240.199} C_VEL
LIN {X 0,Y 551.96,Z 777.902,A -85,B 0,C 180,E1 -2242.298,E2 -2242.298} C_VEL
LIN {X 0,Y 551.921,Z 783.145,A -85,B 0,C 180,E1 -2244.387,E2 -2244.387} C_VEL
LIN {X 0,Y 551.904,Z 786.711,A -85,B 0,C 180,E1 -2246.47,E2 -2246.47} C_VEL
LIN {X 0,Y 551.9,Z 788.575,A -85,B 0,C 180,E1 -2248.548,E2 -2248.548} C_VEL
LIN {X 0,Y 551.902,Z 788.873,A -85,B 0,C 180,E1 -2250.624,E2 -2250.624} C_VEL
LIN {X 0,Y 551.911,Z 787.504,A -85,B 0,C 180,E1 -2252.805,E2 -2252.805} C_VEL
LIN {X 0,Y 551.92,Z 784.578,A -85,B 0,C 180,E1 -2254.885,E2 -2254.885} C_VEL
LIN {X 0,Y 551.938,Z 779.972,A -85,B 0,C 180,E1 -2256.972,E2 -2256.972} C_VEL
LIN {X 0,Y 551.987,Z 773.909,A -85,B 0,C 180,E1 -2258.963,E2 -2258.963} C_VEL
LIN {X 0,Y 552.092,Z 765.953,A -85,B 0,C 180,E1 -2261.014,E2 -2261.014} C_VEL
LIN {X 0,Y 552.263,Z 756.56,A -85,B 0,C 180,E1 -2262.974,E2 -2262.974} C_VEL
LIN {X 0,Y 552.522,Z 745.371,A -85,B 0,C 180,E1 -2264.909,E2 -2264.909} C_VEL
LIN {X 0,Y 552.877,Z 732.126,A -85,B 0,C 180,E1 -2266.82,E2 -2266.82} C_VEL
LIN {X 0,Y 553.325,Z 717.313,A -85,B 0,C 180,E1 -2268.618,E2 -2268.618} C_VEL
LIN {X 0,Y 553.854,Z 701.041,A -85,B 0,C 180,E1 -2270.281,E2 -2270.281} C_VEL
LIN {X 0,Y 554.433,Z 683.855,A -85,B 0,C 180,E1 -2271.76,E2 -2271.76} C_VEL
LIN {X 0,Y 555.015,Z 666.503,A -85,B 0,C 180,E1 -2273.013,E2 -2273.013} C_VEL
LIN {X 0,Y 555.592,Z 648.265,A -85,B 0,C 180,E1 -2274.112,E2 -2274.112} C_VEL
LIN {X 0,Y 556.121,Z 629.25,A -85,B 0,C 180,E1 -2275.051,E2 -2275.051} C_VEL
LIN {X 0,Y 556.633,Z 609.344,A -85,B 0,C 180,E1 -2275.824,E2 -2275.824} C_VEL
LIN {X 0,Y 557.07,Z 588.839,A -85,B 0,C 180,E1 -2276.415,E2 -2276.415} C_VEL
LIN {X 0,Y 557.318,Z 567.71,A -85,B 0,C 180,E1 -2276.816,E2 -2276.816} C_VEL
LIN {X 0,Y 558.686,Z 334.299,A -85,B 0,C 180,E1 -2280.091,E2 -2280.091} C_VEL
LIN {X 0,Y 558.522,Z 323.011,A -85,B 0,C 180,E1 -2280.265,E2 -2280.265} C_VEL
LIN {X 0,Y 557.204,Z 314.837,A -85,B 0,C 180,E1 -2280.49,E2 -2280.49} C_VEL
LIN {X 0,Y 557.862,Z 282.456,A -85,B 0,C 180,E1 -2282.755,E2 -2282.755} C_VEL
LIN {X 0,Y 552.372,Z 267.996,A -85,B 0,C 180,E1 -2284.167,E2 -2284.167} C_VEL
LIN {X 0,Y 552.332,Z 267.687,A -85,B 0,C 180,E1 -2285.147,E2 -2285.147} C_VEL
LIN {X 0,Y 552.345,Z 267.684,A -85,B 0,C 180,E1 -2288.555,E2 -2288.555} C_VEL
LIN {X 0,Y 552.304,Z 267.686,A -85,B 0,C 180,E1 -2291.776,E2 -2291.776} C_VEL
LIN {X 0,Y 552.336,Z 267.688,A -85,B 0,C 180,E1 -2295.091,E2 -2295.091} C_VEL
LIN {X 0,Y 552.327,Z 267.683,A -85,B 0,C 180,E1 -2298.387,E2 -2298.387} C_VEL
LIN {X 0,Y 552.298,Z 267.688,A -85,B 0,C 180,E1 -2301.619,E2 -2301.619} C_VEL
LIN {X 0,Y 552.345,Z 267.686,A -85,B 0,C 180,E1 -2304.907,E2 -2304.907} C_VEL
LIN {X 0,Y 552.319,Z 267.821,A -85,B 0,C 180,E1 -2308.181,E2 -2308.181} C_VEL
LIN {X 0,Y 552.771,Z 269.52,A -85,B 0,C 180,E1 -2308.425,E2 -2308.425} C_VEL
LIN {X 0,Y 556.692,Z 281.727,A -85,B 0,C 180,E1 -2309.689,E2 -2309.689} C_VEL
LIN {X 0,Y 555.725,Z 323.491,A -85,B 0,C 180,E1 -2313.038,E2 -2313.038} C_VEL
LIN {X 0,Y 555.391,Z 342.331,A -85,B 0,C 180,E1 -2314.502,E2 -2314.502} C_VEL
LIN {X 0,Y 556.752,Z 351.91,A -85,B 0,C 180,E1 -2314.716,E2 -2314.716} C_VEL
LIN {X 0,Y 555.703,Z 559.825,A -85,B 0,C 180,E1 -2317.574,E2 -2317.574} C_VEL
LIN {X 0,Y 555.419,Z 579.56,A -85,B 0,C 180,E1 -2318.045,E2 -2318.045} C_VEL
LIN {X 0,Y 555.062,Z 598.233,A -85,B 0,C 180,E1 -2318.69,E2 -2318.69} C_VEL
LIN {X 0,Y 554.625,Z 616.494,A -85,B 0,C 180,E1 -2319.529,E2 -2319.529} C_VEL
LIN {X 0,Y 554.16,Z 634.188,A -85,B 0,C 180,E1 -2320.556,E2 -2320.556} C_VEL
LIN {X 0,Y 553.694,Z 650.84,A -85,B 0,C 180,E1 -2321.747,E2 -2321.747} C_VEL
LIN {X 0,Y 553.251,Z 666.265,A -85,B 0,C 180,E1 -2323.085,E2 -2323.085} C_VEL
LIN {X 0,Y 552.858,Z 680.646,A -85,B 0,C 180,E1 -2324.583,E2 -2324.583} C_VEL
LIN {X 0,Y 552.542,Z 693.493,A -85,B 0,C 180,E1 -2326.181,E2 -2326.181} C_VEL
LIN {X 0,Y 552.293,Z 704.824,A -85,B 0,C 180,E1 -2327.878,E2 -2327.878} C_VEL
LIN {X 0,Y 552.12,Z 714.658,A -85,B 0,C 180,E1 -2329.672,E2 -2329.672} C_VEL
LIN {X 0,Y 552.001,Z 722.972,A -85,B 0,C 180,E1 -2331.564,E2 -2331.564} C_VEL
LIN {X 0,Y 551.942,Z 729.719,A -85,B 0,C 180,E1 -2333.552,E2 -2333.552} C_VEL
LIN {X 0,Y 551.914,Z 734.549,A -85,B 0,C 180,E1 -2335.533,E2 -2335.533} C_VEL
LIN {X 0,Y 551.913,Z 737.578,A -85,B 0,C 180,E1 -2337.508,E2 -2337.508} C_VEL
LIN {X 0,Y 551.909,Z 738.886,A -85,B 0,C 180,E1 -2339.481,E2 -2339.481} C_VEL
LIN {X 0,Y 551.911,Z 738.468,A -85,B 0,C 180,E1 -2341.558,E2 -2341.558} C_VEL
LIN {X 0,Y 551.91,Z 736.34,A -85,B 0,C 180,E1 -2343.532,E2 -2343.532} C_VEL
LIN {X 0,Y 551.928,Z 732.456,A -85,B 0,C 180,E1 -2345.51,E2 -2345.51} C_VEL
LIN {X 0,Y 551.965,Z 726.721,A -85,B 0,C 180,E1 -2347.495,E2 -2347.495} C_VEL
LIN {X 0,Y 552.061,Z 718.994,A -85,B 0,C 180,E1 -2349.487,E2 -2349.487} C_VEL
LIN {X 0,Y 552.207,Z 709.621,A -85,B 0,C 180,E1 -2351.383,E2 -2351.383} C_VEL
LIN {X 0,Y 552.424,Z 698.615,A -85,B 0,C 180,E1 -2353.183,E2 -2353.183} C_VEL
LIN {X 0,Y 552.725,Z 685.961,A -85,B 0,C 180,E1 -2354.885,E2 -2354.885} C_VEL
LIN {X 0,Y 553.089,Z 672.079,A -85,B 0,C 180,E1 -2356.435,E2 -2356.435} C_VEL
LIN {X 0,Y 553.514,Z 657.117,A -85,B 0,C 180,E1 -2357.83,E2 -2357.83} C_VEL
LIN {X 0,Y 553.984,Z 640.418,A -85,B 0,C 180,E1 -2359.115,E2 -2359.115} C_VEL
LIN {X 0,Y 554.455,Z 623.149,A -85,B 0,C 180,E1 -2360.203,E2 -2360.203} C_VEL
LIN {X 0,Y 554.885,Z 606.004,A -85,B 0,C 180,E1 -2361.069,E2 -2361.069} C_VEL
LIN {X 0,Y 555.124,Z 594.384,A -85,B 0,C 180,E1 -2361.548,E2 -2361.548} C_VEL
LIN {X 0,Y 554.33,Z 587.206,A -85,B 0,C 180,E1 -2361.846,E2 -2361.846} C_VEL
LIN {X 0,Y 549.287,Z 570.234,A -85,B 0,C 180,E1 -2362.561,E2 -2362.561} C_VEL
LIN {X 0,Y 548.272,Z 562.843,A -85,B 0,C 180,E1 -2362.775,E2 -2362.775} C_VEL
LIN {X 0,Y 548.266,Z 561.759,A -85,B 0,C 180,E1 -2362.798,E2 -2362.798} C_VEL
LIN {X 0,Y 548.538,Z 526.374,A -85,B 0,C 180,E1 -2363.322,E2 -2363.322} C_VEL
LIN {X 0,Y 549.356,Z 350.631,A -85,B 0,C 180,E1 -2365.758,E2 -2365.758} C_VEL
LIN {X 0,Y 547.921,Z 342.045,A -85,B 0,C 180,E1 -2365.974,E2 -2365.974} C_VEL
LIN {X 0,Y 548.988,Z 299.37,A -85,B 0,C 180,E1 -2369.396,E2 -2369.396} C_VEL
LIN {X 0,Y 549.296,Z 283.514,A -85,B 0,C 180,E1 -2370.703,E2 -2370.703} C_VEL
LIN {X 0,Y 544.384,Z 268.893,A -85,B 0,C 180,E1 -2372.309,E2 -2372.309} C_VEL
LIN {X 0,Y 544.401,Z 268.658,A -85,B 0,C 180,E1 -2375.348,E2 -2375.348} C_VEL
LIN {X 0,Y 544.398,Z 268.676,A -85,B 0,C 180,E1 -2378.778,E2 -2378.778} C_VEL
LIN {X 0,Y 544.374,Z 268.67,A -85,B 0,C 180,E1 -2382.099,E2 -2382.099} C_VEL
LIN {X 0,Y 544.403,Z 268.669,A -85,B 0,C 180,E1 -2385.448,E2 -2385.448} C_VEL
LIN {X 0,Y 544.397,Z 268.674,A -85,B 0,C 180,E1 -2388.889,E2 -2388.889} C_VEL
LIN {X 0,Y 544.393,Z 268.674,A -85,B 0,C 180,E1 -2392.294,E2 -2392.294} C_VEL
LIN {X 0,Y 544.402,Z 268.668,A -85,B 0,C 180,E1 -2395.74,E2 -2395.74} C_VEL
LIN {X 0,Y 544.377,Z 268.67,A -85,B 0,C 180,E1 -2399.065,E2 -2399.065} C_VEL
LIN {X 0,Y 544.397,Z 268.677,A -85,B 0,C 180,E1 -2402.429,E2 -2402.429} C_VEL
LIN {X 0,Y 544.403,Z 268.666,A -85,B 0,C 180,E1 -2405.822,E2 -2405.822} C_VEL
LIN {X 0,Y 544.358,Z 268.671,A -85,B 0,C 180,E1 -2409.124,E2 -2409.124} C_VEL
LIN {X 0,Y 544.37,Z 268.677,A -85,B 0,C 180,E1 -2412.468,E2 -2412.468} C_VEL
LIN {X 0,Y 544.378,Z 268.661,A -85,B 0,C 180,E1 -2415.643,E2 -2415.643} C_VEL
LIN {X 0,Y 544.332,Z 268.675,A -85,B 0,C 180,E1 -2418.879,E2 -2418.879} C_VEL
LIN {X 0,Y 544.35,Z 268.818,A -85,B 0,C 180,E1 -2421.191,E2 -2421.191} C_VEL
LIN {X 0,Y 545.018,Z 271.044,A -85,B 0,C 180,E1 -2421.453,E2 -2421.453} C_VEL
LIN {X 0,Y 548.268,Z 282.133,A -85,B 0,C 180,E1 -2422.507,E2 -2422.507} C_VEL
LIN {X 0,Y 548.042,Z 321.72,A -85,B 0,C 180,E1 -2425.604,E2 -2425.604} C_VEL
LIN {X 0,Y 547.589,Z 362.631,A -85,B 0,C 180,E1 -2428.796,E2 -2428.796} C_VEL
LIN {X 0,Y 546.939,Z 404.882,A -85,B 0,C 180,E1 -2432.094,E2 -2432.094} C_VEL
LIN {X 0,Y 546.175,Z 447.44,A -85,B 0,C 180,E1 -2435.409,E2 -2435.409} C_VEL
LIN {X 0,Y 545.823,Z 472.822,A -85,B 0,C 180,E1 -2437.35,E2 -2437.35} C_VEL
LIN {X 0,Y 546.547,Z 481.441,A -85,B 0,C 180,E1 -2437.498,E2 -2437.498} C_VEL
LIN {X 0,Y 545.989,Z 615.312,A -85,B 0,C 180,E1 -2439.309,E2 -2439.309} C_VEL
LIN {X 0,Y 545.815,Z 631.31,A -85,B 0,C 180,E1 -2439.719,E2 -2439.719} C_VEL
LIN {X 0,Y 545.557,Z 647.511,A -85,B 0,C 180,E1 -2440.346,E2 -2440.346} C_VEL
LIN {X 0,Y 545.268,Z 661.83,A -85,B 0,C 180,E1 -2441.1,E2 -2441.1} C_VEL
LIN {X 0,Y 544.939,Z 676.127,A -85,B 0,C 180,E1 -2442.072,E2 -2442.072} C_VEL
LIN {X 0,Y 544.665,Z 688.782,A -85,B 0,C 180,E1 -2443.156,E2 -2443.156} C_VEL
LIN {X 0,Y 544.4,Z 700.969,A -85,B 0,C 180,E1 -2444.463,E2 -2444.463} C_VEL
LIN {X 0,Y 544.21,Z 710.834,A -85,B 0,C 180,E1 -2445.777,E2 -2445.777} C_VEL
LIN {X 0,Y 544.061,Z 720.003,A -85,B 0,C 180,E1 -2447.319,E2 -2447.319} C_VEL
LIN {X 0,Y 543.978,Z 727.166,A -85,B 0,C 180,E1 -2448.873,E2 -2448.873} C_VEL
LIN {X 0,Y 543.931,Z 732.813,A -85,B 0,C 180,E1 -2450.553,E2 -2450.553} C_VEL
LIN {X 0,Y 543.922,Z 736.644,A -85,B 0,C 180,E1 -2452.25,E2 -2452.25} C_VEL
LIN {X 0,Y 543.916,Z 738.634,A -85,B 0,C 180,E1 -2453.989,E2 -2453.989} C_VEL
LIN {X 0,Y 543.916,Z 738.853,A -85,B 0,C 180,E1 -2455.742,E2 -2455.742} C_VEL
LIN {X 0,Y 543.917,Z 737.184,A -85,B 0,C 180,E1 -2457.476,E2 -2457.476} C_VEL
LIN {X 0,Y 543.932,Z 733.808,A -85,B 0,C 180,E1 -2459.172,E2 -2459.172} C_VEL
LIN {X 0,Y 543.964,Z 728.552,A -85,B 0,C 180,E1 -2460.851,E2 -2460.851} C_VEL
LIN {X 0,Y 544.043,Z 721.506,A -85,B 0,C 180,E1 -2462.481,E2 -2462.481} C_VEL
LIN {X 0,Y 544.17,Z 713.158,A -85,B 0,C 180,E1 -2463.955,E2 -2463.955} C_VEL
LIN {X 0,Y 544.363,Z 702.783,A -85,B 0,C 180,E1 -2465.407,E2 -2465.407} C_VEL
LIN {X 0,Y 544.611,Z 691.264,A -85,B 0,C 180,E1 -2466.689,E2 -2466.689} C_VEL
LIN {X 0,Y 544.895,Z 678.555,A -85,B 0,C 180,E1 -2467.829,E2 -2467.829} C_VEL
LIN {X 0,Y 545.193,Z 665.066,A -85,B 0,C 180,E1 -2468.791,E2 -2468.791} C_VEL
LIN {X 0,Y 545.503,Z 649.951,A -85,B 0,C 180,E1 -2469.63,E2 -2469.63} C_VEL
LIN {X 0,Y 545.777,Z 634.463,A -85,B 0,C 180,E1 -2470.266,E2 -2470.266} C_VEL
LIN {X 0,Y 545.961,Z 617.574,A -85,B 0,C 180,E1 -2470.736,E2 -2470.736} C_VEL
LIN {X 0,Y 546.08,Z 591.808,A -85,B 0,C 180,E1 -2471.122,E2 -2471.122} C_VEL
LIN {X 0,Y 546.334,Z 477.199,A -85,B 0,C 180,E1 -2472.656,E2 -2472.656} C_VEL
LIN {X 0,Y 545.789,Z 472.587,A -85,B 0,C 180,E1 -2472.755,E2 -2472.755} C_VEL
LIN {X 0,Y 546.359,Z 437.042,A -85,B 0,C 180,E1 -2475.5,E2 -2475.5} C_VEL
LIN {X 0,Y 547.126,Z 394.245,A -85,B 0,C 180,E1 -2478.86,E2 -2478.86} C_VEL
LIN {X 0,Y 547.621,Z 354.566,A -85,B 0,C 180,E1 -2481.893,E2 -2481.893} C_VEL
LIN {X 0,Y 547.909,Z 314.541,A -85,B 0,C 180,E1 -2484.975,E2 -2484.975} C_VEL
LIN {X 0,Y 547.813,Z 280.315,A -85,B 0,C 180,E1 -2487.609,E2 -2487.609} C_VEL
LIN {X 0,Y 544.436,Z 268.93,A -85,B 0,C 180,E1 -2488.685,E2 -2488.685} C_VEL
LIN {X 0,Y 544.369,Z 268.677,A -85,B 0,C 180,E1 -2491.836,E2 -2491.836} C_VEL
LIN {X 0,Y 544.362,Z 268.675,A -85,B 0,C 180,E1 -2495.242,E2 -2495.242} C_VEL
LIN {X 0,Y 544.406,Z 268.671,A -85,B 0,C 180,E1 -2498.562,E2 -2498.562} C_VEL
LIN {X 0,Y 544.369,Z 268.673,A -85,B 0,C 180,E1 -2501.916,E2 -2501.916} C_VEL
LIN {X 0,Y 544.364,Z 268.671,A -85,B 0,C 180,E1 -2505.317,E2 -2505.317} C_VEL
LIN {X 0,Y 544.404,Z 268.673,A -85,B 0,C 180,E1 -2508.559,E2 -2508.559} C_VEL
LIN {X 0,Y 544.363,Z 268.674,A -85,B 0,C 180,E1 -2511.88,E2 -2511.88} C_VEL
LIN {X 0,Y 544.369,Z 268.671,A -85,B 0,C 180,E1 -2515.364,E2 -2515.364} C_VEL
LIN {X 0,Y 544.405,Z 268.674,A -85,B 0,C 180,E1 -2518.631,E2 -2518.631} C_VEL
LIN {X 0,Y 544.363,Z 268.672,A -85,B 0,C 180,E1 -2521.894,E2 -2521.894} C_VEL
LIN {X 0,Y 544.385,Z 268.67,A -85,B 0,C 180,E1 -2525.269,E2 -2525.269} C_VEL
LIN {X 0,Y 544.406,Z 268.673,A -85,B 0,C 180,E1 -2528.661,E2 -2528.661} C_VEL
LIN {X 0,Y 544.365,Z 268.673,A -85,B 0,C 180,E1 -2531.979,E2 -2531.979} C_VEL
LIN {X 0,Y 544.386,Z 268.668,A -85,B 0,C 180,E1 -2535.373,E2 -2535.373} C_VEL
LIN {X 0,Y 544.403,Z 268.673,A -85,B 0,C 180,E1 -2538.748,E2 -2538.748} C_VEL
LIN {X 0,Y 544.364,Z 268.672,A -85,B 0,C 180,E1 -2542.005,E2 -2542.005} C_VEL
LIN {X 0,Y 544.395,Z 268.669,A -85,B 0,C 180,E1 -2545.365,E2 -2545.365} C_VEL
LIN {X 0,Y 544.403,Z 268.675,A -85,B 0,C 180,E1 -2548.763,E2 -2548.763} C_VEL
LIN {X 0,Y 544.367,Z 268.672,A -85,B 0,C 180,E1 -2552.06,E2 -2552.06} C_VEL
LIN {X 0,Y 544.402,Z 268.668,A -85,B 0,C 180,E1 -2555.37,E2 -2555.37} C_VEL
LIN {X 0,Y 544.403,Z 268.676,A -85,B 0,C 180,E1 -2558.776,E2 -2558.776} C_VEL
LIN {X 0,Y 544.369,Z 268.673,A -85,B 0,C 180,E1 -2562.098,E2 -2562.098} C_VEL
LIN {X 0,Y 544.403,Z 268.669,A -85,B 0,C 180,E1 -2565.448,E2 -2565.448} C_VEL
LIN {X 0,Y 544.404,Z 268.675,A -85,B 0,C 180,E1 -2568.892,E2 -2568.892} C_VEL
LIN {X 0,Y 544.369,Z 268.676,A -85,B 0,C 180,E1 -2572.166,E2 -2572.166} C_VEL
LIN {X 0,Y 544.429,Z 268.872,A -85,B 0,C 180,E1 -2575.299,E2 -2575.299} C_VEL
LIN {X 0,Y 546.406,Z 274.424,A -85,B 0,C 180,E1 -2575.896,E2 -2575.896} C_VEL
LIN {X 0,Y 550.825,Z 286.317,A -85,B 0,C 180,E1 -2577.063,E2 -2577.063} C_VEL
LIN {X 0,Y 550.139,Z 315.757,A -85,B 0,C 180,E1 -2579.113,E2 -2579.113} C_VEL
LIN {X 0,Y 551.816,Z 326.941,A -85,B 0,C 180,E1 -2579.386,E2 -2579.386} C_VEL
LIN {X 0,Y 550.262,Z 556.513,A -85,B 0,C 180,E1 -2582.648,E2 -2582.648} C_VEL
LIN {X 0,Y 549.951,Z 582.995,A -85,B 0,C 180,E1 -2583.084,E2 -2583.084} C_VEL
LIN {X 0,Y 549.528,Z 603.787,A -85,B 0,C 180,E1 -2583.631,E2 -2583.631} C_VEL
LIN {X 0,Y 549.038,Z 622.887,A -85,B 0,C 180,E1 -2584.317,E2 -2584.317} C_VEL
LIN {X 0,Y 548.397,Z 642.486,A -85,B 0,C 180,E1 -2585.226,E2 -2585.226} C_VEL
LIN {X 0,Y 547.724,Z 661.447,A -85,B 0,C 180,E1 -2586.323,E2 -2586.323} C_VEL
LIN {X 0,Y 547.025,Z 679.674,A -85,B 0,C 180,E1 -2587.6,E2 -2587.6} C_VEL
LIN {X 0,Y 546.345,Z 696.844,A -85,B 0,C 180,E1 -2589.037,E2 -2589.037} C_VEL
LIN {X 0,Y 545.715,Z 713.203,A -85,B 0,C 180,E1 -2590.662,E2 -2590.662} C_VEL
LIN {X 0,Y 545.178,Z 727.917,A -85,B 0,C 180,E1 -2592.387,E2 -2592.387} C_VEL
LIN {X 0,Y 544.771,Z 740.579,A -85,B 0,C 180,E1 -2594.131,E2 -2594.131} C_VEL
LIN {X 0,Y 544.432,Z 752.54,A -85,B 0,C 180,E1 -2596.08,E2 -2596.08} C_VEL
LIN {X 0,Y 544.187,Z 762.914,A -85,B 0,C 180,E1 -2598.126,E2 -2598.126} C_VEL
LIN {X 0,Y 544.047,Z 771.283,A -85,B 0,C 180,E1 -2600.16,E2 -2600.16} C_VEL
LIN {X 0,Y 543.966,Z 778.205,A -85,B 0,C 180,E1 -2602.29,E2 -2602.29} C_VEL
LIN {X 0,Y 543.921,Z 783.351,A -85,B 0,C 180,E1 -2604.41,E2 -2604.41} C_VEL
LIN {X 0,Y 543.903,Z 786.829,A -85,B 0,C 180,E1 -2606.523,E2 -2606.523} C_VEL
LIN {X 0,Y 543.9,Z 788.642,A -85,B 0,C 180,E1 -2608.632,E2 -2608.632} C_VEL
LIN {X 0,Y 543.906,Z 788.851,A -85,B 0,C 180,E1 -2610.738,E2 -2610.738} C_VEL
LIN {X 0,Y 543.91,Z 787.393,A -85,B 0,C 180,E1 -2612.952,E2 -2612.952} C_VEL
LIN {X 0,Y 543.914,Z 784.373,A -85,B 0,C 180,E1 -2615.063,E2 -2615.063} C_VEL
LIN {X 0,Y 543.941,Z 779.709,A -85,B 0,C 180,E1 -2617.182,E2 -2617.182} C_VEL
LIN {X 0,Y 544.01,Z 773.367,A -85,B 0,C 180,E1 -2619.259,E2 -2619.259} C_VEL
LIN {X 0,Y 544.134,Z 765.716,A -85,B 0,C 180,E1 -2621.233,E2 -2621.233} C_VEL
LIN {X 0,Y 544.347,Z 755.986,A -85,B 0,C 180,E1 -2623.275,E2 -2623.275} C_VEL
LIN {X 0,Y 544.646,Z 744.783,A -85,B 0,C 180,E1 -2625.221,E2 -2625.221} C_VEL
LIN {X 0,Y 545.063,Z 731.768,A -85,B 0,C 180,E1 -2627.115,E2 -2627.115} C_VEL
LIN {X 0,Y 545.57,Z 717.476,A -85,B 0,C 180,E1 -2628.874,E2 -2628.874} C_VEL
LIN {X 0,Y 546.181,Z 701.37,A -85,B 0,C 180,E1 -2630.547,E2 -2630.547} C_VEL
LIN {X 0,Y 546.853,Z 684.004,A -85,B 0,C 180,E1 -2632.065,E2 -2632.065} C_VEL
LIN {X 0,Y 547.526,Z 666.499,A -85,B 0,C 180,E1 -2633.346,E2 -2633.346} C_VEL
LIN {X 0,Y 548.212,Z 647.865,A -85,B 0,C 180,E1 -2634.481,E2 -2634.481} C_VEL
LIN {X 0,Y 548.858,Z 627.964,A -85,B 0,C 180,E1 -2635.464,E2 -2635.464} C_VEL
LIN {X 0,Y 549.414,Z 607.739,A -85,B 0,C 180,E1 -2636.243,E2 -2636.243} C_VEL
LIN {X 0,Y 549.907,Z 587.593,A -85,B 0,C 180,E1 -2636.815,E2 -2636.815} C_VEL
LIN {X 0,Y 550.198,Z 566.503,A -85,B 0,C 180,E1 -2637.212,E2 -2637.212} C_VEL
LIN {X 0,Y 551.769,Z 333.79,A -85,B 0,C 180,E1 -2640.515,E2 -2640.515} C_VEL
LIN {X 0,Y 551.592,Z 324.232,A -85,B 0,C 180,E1 -2640.668,E2 -2640.668} C_VEL
LIN {X 0,Y 550.068,Z 315.089,A -85,B 0,C 180,E1 -2640.913,E2 -2640.913} C_VEL
LIN {X 0,Y 550.7,Z 285.522,A -85,B 0,C 180,E1 -2642.985,E2 -2642.985} C_VEL
LIN {X 0,Y 544.476,Z 269.148,A -85,B 0,C 180,E1 -2644.573,E2 -2644.573} C_VEL
LIN {X 0,Y 544.404,Z 268.675,A -85,B 0,C 180,E1 -2645.003,E2 -2645.003} C_VEL
LIN {X 0,Y 544.399,Z 268.673,A -85,B 0,C 180,E1 -2648.374,E2 -2648.374} C_VEL
LIN {X 0,Y 544.366,Z 268.676,A -85,B 0,C 180,E1 -2651.675,E2 -2651.675} C_VEL
LIN {X 0,Y 544.401,Z 268.676,A -85,B 0,C 180,E1 -2655.001,E2 -2655.001} C_VEL
LIN {X 0,Y 544.388,Z 268.673,A -85,B 0,C 180,E1 -2658.377,E2 -2658.377} C_VEL
LIN {X 0,Y 544.358,Z 268.677,A -85,B 0,C 180,E1 -2661.657,E2 -2661.657} C_VEL
LIN {X 0,Y 544.404,Z 268.676,A -85,B 0,C 180,E1 -2664.999,E2 -2664.999} C_VEL
LIN {X 0,Y 544.389,Z 268.94,A -85,B 0,C 180,E1 -2667.755,E2 -2667.755} C_VEL
LIN {X 0,Y 548.234,Z 280.298,A -85,B 0,C 180,E1 -2669.049,E2 -2669.049} C_VEL
LIN {X 0,Y 549.396,Z 284.616,A -85,B 0,C 180,E1 -2669.486,E2 -2669.486} C_VEL
LIN {X 0,Y 548.278,Z 326.381,A -85,B 0,C 180,E1 -2672.877,E2 -2672.877} C_VEL
LIN {X 0,Y 547.947,Z 342.348,A -85,B 0,C 180,E1 -2674.13,E2 -2674.13} C_VEL
LIN {X 0,Y 549.515,Z 352.978,A -85,B 0,C 180,E1 -2674.373,E2 -2674.373} C_VEL
LIN {X 0,Y 548.308,Z 559.851,A -85,B 0,C 180,E1 -2677.254,E2 -2677.254} C_VEL
LIN {X 0,Y 547.981,Z 579.575,A -85,B 0,C 180,E1 -2677.732,E2 -2677.732} C_VEL
LIN {X 0,Y 547.57,Z 598.25,A -85,B 0,C 180,E1 -2678.384,E2 -2678.384} C_VEL
LIN {X 0,Y 547.067,Z 616.503,A -85,B 0,C 180,E1 -2679.233,E2 -2679.233} C_VEL
LIN {X 0,Y 546.527,Z 634.25,A -85,B 0,C 180,E1 -2680.277,E2 -2680.277} C_VEL
LIN {X 0,Y 545.994,Z 650.785,A -85,B 0,C 180,E1 -2681.475,E2 -2681.475} C_VEL
LIN {X 0,Y 545.477,Z 666.271,A -85,B 0,C 180,E1 -2682.836,E2 -2682.836} C_VEL
LIN {X 0,Y 545.009,Z 681.023,A -85,B 0,C 180,E1 -2684.399,E2 -2684.399} C_VEL
LIN {X 0,Y 544.633,Z 694.276,A -85,B 0,C 180,E1 -2686.085,E2 -2686.085} C_VEL
LIN {X 0,Y 544.348,Z 705.47,A -85,B 0,C 180,E1 -2687.806,E2 -2687.806} C_VEL
LIN {X 0,Y 544.148,Z 715.181,A -85,B 0,C 180,E1 -2689.626,E2 -2689.626} C_VEL
LIN {X 0,Y 544.013,Z 723.379,A -85,B 0,C 180,E1 -2691.545,E2 -2691.545} C_VEL
LIN {X 0,Y 543.947,Z 730.024,A -85,B 0,C 180,E1 -2693.562,E2 -2693.562} C_VEL
LIN {X 0,Y 543.916,Z 734.758,A -85,B 0,C 180,E1 -2695.572,E2 -2695.572} C_VEL
LIN {X 0,Y 543.913,Z 737.693,A -85,B 0,C 180,E1 -2697.577,E2 -2697.577} C_VEL
LIN {X 0,Y 543.906,Z 738.908,A -85,B 0,C 180,E1 -2699.579,E2 -2699.579} C_VEL
LIN {X 0,Y 543.91,Z 738.4,A -85,B 0,C 180,E1 -2701.686,E2 -2701.686} C_VEL
LIN {X 0,Y 543.909,Z 736.184,A -85,B 0,C 180,E1 -2703.689,E2 -2703.689} C_VEL
LIN {X 0,Y 543.934,Z 732.204,A -85,B 0,C 180,E1 -2705.697,E2 -2705.697} C_VEL
LIN {X 0,Y 543.974,Z 726.72,A -85,B 0,C 180,E1 -2707.605,E2 -2707.605} C_VEL
LIN {X 0,Y 544.085,Z 718.991,A -85,B 0,C 180,E1 -2709.627,E2 -2709.627} C_VEL
LIN {X 0,Y 544.26,Z 709.62,A -85,B 0,C 180,E1 -2711.552,E2 -2711.552} C_VEL
LIN {X 0,Y 544.515,Z 698.615,A -85,B 0,C 180,E1 -2713.378,E2 -2713.378} C_VEL
LIN {X 0,Y 544.866,Z 685.958,A -85,B 0,C 180,E1 -2715.105,E2 -2715.105} C_VEL
LIN {X 0,Y 545.3,Z 671.961,A -85,B 0,C 180,E1 -2716.688,E2 -2716.688} C_VEL
LIN {X 0,Y 545.786,Z 657.173,A -85,B 0,C 180,E1 -2718.085,E2 -2718.085} C_VEL
LIN {X 0,Y 546.31,Z 641.073,A -85,B 0,C 180,E1 -2719.346,E2 -2719.346} C_VEL
LIN {X 0,Y 546.844,Z 624.073,A -85,B 0,C 180,E1 -2720.441,E2 -2720.441} C_VEL
LIN {X 0,Y 547.365,Z 605.986,A -85,B 0,C 180,E1 -2721.372,E2 -2721.372} C_VEL
LIN {X 0,Y 547.825,Z 587.15,A -85,B 0,C 180,E1 -2722.117,E2 -2722.117} C_VEL
LIN {X 0,Y 548.195,Z 567.733,A -85,B 0,C 180,E1 -2722.672,E2 -2722.672} C_VEL
LIN {X 0,Y 548.266,Z 561.759,A -85,B 0,C 180,E1 -2722.798,E2 -2722.798} C_VEL
LIN {X 0,Y 547.467,Z 554.222,A -85,B 0,C 180,E1 -2722.975,E2 -2722.975} C_VEL
LIN {X 0,Y 541.849,Z 534.391,A -85,B 0,C 180,E1 -2723.516,E2 -2723.516} C_VEL
LIN {X 0,Y 541.182,Z 527.864,A -85,B 0,C 180,E1 -2723.636,E2 -2723.636} C_VEL
LIN {X 0,Y 542.134,Z 351.748,A -85,B 0,C 180,E1 -2726.11,E2 -2726.11} C_VEL
LIN {X 0,Y 540.5,Z 342.045,A -85,B 0,C 180,E1 -2726.358,E2 -2726.358} C_VEL
LIN {X 0,Y 541.733,Z 299.305,A -85,B 0,C 180,E1 -2729.834,E2 -2729.834} C_VEL
LIN {X 0,Y 541.998,Z 286.28,A -85,B 0,C 180,E1 -2730.927,E2 -2730.927} C_VEL
LIN {X 0,Y 536.481,Z 269.937,A -85,B 0,C 180,E1 -2732.753,E2 -2732.753} C_VEL
LIN {X 0,Y 536.419,Z 269.631,A -85,B 0,C 180,E1 -2734.387,E2 -2734.387} C_VEL
LIN {X 0,Y 536.435,Z 269.661,A -85,B 0,C 180,E1 -2737.823,E2 -2737.823} C_VEL
LIN {X 0,Y 536.464,Z 269.659,A -85,B 0,C 180,E1 -2741.151,E2 -2741.151} C_VEL
LIN {X 0,Y 536.456,Z 269.662,A -85,B 0,C 180,E1 -2744.603,E2 -2744.603} C_VEL
LIN {X 0,Y 536.445,Z 269.661,A -85,B 0,C 180,E1 -2748.047,E2 -2748.047} C_VEL
LIN {X 0,Y 536.465,Z 269.657,A -85,B 0,C 180,E1 -2751.5,E2 -2751.5} C_VEL
LIN {X 0,Y 536.447,Z 269.661,A -85,B 0,C 180,E1 -2754.965,E2 -2754.965} C_VEL
LIN {X 0,Y 536.464,Z 269.665,A -85,B 0,C 180,E1 -2758.417,E2 -2758.417} C_VEL
LIN {X 0,Y 536.464,Z 269.656,A -85,B 0,C 180,E1 -2761.865,E2 -2761.865} C_VEL
LIN {X 0,Y 536.43,Z 269.656,A -85,B 0,C 180,E1 -2765.204,E2 -2765.204} C_VEL
LIN {X 0,Y 536.427,Z 269.661,A -85,B 0,C 180,E1 -2768.686,E2 -2768.686} C_VEL
LIN {X 0,Y 536.466,Z 269.659,A -85,B 0,C 180,E1 -2771.977,E2 -2771.977} C_VEL
LIN {X 0,Y 536.406,Z 269.656,A -85,B 0,C 180,E1 -2775.204,E2 -2775.204} C_VEL
LIN {X 0,Y 536.398,Z 269.665,A -85,B 0,C 180,E1 -2778.712,E2 -2778.712} C_VEL
LIN {X 0,Y 536.424,Z 269.919,A -85,B 0,C 180,E1 -2780.856,E2 -2780.856} C_VEL
LIN {X 0,Y 540.848,Z 284.151,A -85,B 0,C 180,E1 -2782.267,E2 -2782.267} C_VEL
LIN {X 0,Y 540.57,Z 322.999,A -85,B 0,C 180,E1 -2785.331,E2 -2785.331} C_VEL
LIN {X 0,Y 540.041,Z 364.148,A -85,B 0,C 180,E1 -2788.567,E2 -2788.567} C_VEL
LIN {X 0,Y 539.314,Z 406.637,A -85,B 0,C 180,E1 -2791.911,E2 -2791.911} C_VEL
LIN {X 0,Y 538.499,Z 448.804,A -85,B 0,C 180,E1 -2795.219,E2 -2795.219} C_VEL
LIN {X 0,Y 538.099,Z 472.579,A -85,B 0,C 180,E1 -2797.07,E2 -2797.07} C_VEL
LIN {X 0,Y 538.922,Z 482.051,A -85,B 0,C 180,E1 -2797.248,E2 -2797.248} C_VEL
LIN {X 0,Y 538.288,Z 615.431,A -85,B 0,C 180,E1 -2799.08,E2 -2799.08} C_VEL
LIN {X 0,Y 538.091,Z 631.37,A -85,B 0,C 180,E1 -2799.494,E2 -2799.494} C_VEL
LIN {X 0,Y 537.799,Z 647.272,A -85,B 0,C 180,E1 -2800.118,E2 -2800.118} C_VEL
LIN {X 0,Y 537.472,Z 661.659,A -85,B 0,C 180,E1 -2800.883,E2 -2800.883} C_VEL
LIN {X 0,Y 537.098,Z 675.993,A -85,B 0,C 180,E1 -2801.869,E2 -2801.869} C_VEL
LIN {X 0,Y 536.784,Z 688.686,A -85,B 0,C 180,E1 -2802.969,E2 -2802.969} C_VEL
LIN {X 0,Y 536.485,Z 700.671,A -85,B 0,C 180,E1 -2804.27,E2 -2804.27} C_VEL
LIN {X 0,Y 536.251,Z 711.135,A -85,B 0,C 180,E1 -2805.684,E2 -2805.684} C_VEL
LIN {X 0,Y 536.081,Z 720.309,A -85,B 0,C 180,E1 -2807.263,E2 -2807.263} C_VEL
LIN {X 0,Y 535.987,Z 727.339,A -85,B 0,C 180,E1 -2808.826,E2 -2808.826} C_VEL
LIN {X 0,Y 535.933,Z 732.938,A -85,B 0,C 180,E1 -2810.531,E2 -2810.531} C_VEL
LIN {X 0,Y 535.923,Z 736.713,A -85,B 0,C 180,E1 -2812.254,E2 -2812.254} C_VEL
LIN {X 0,Y 535.916,Z 738.649,A -85,B 0,C 180,E1 -2813.997,E2 -2813.997} C_VEL
LIN {X 0,Y 535.915,Z 738.847,A -85,B 0,C 180,E1 -2815.765,E2 -2815.765} C_VEL
LIN {X 0,Y 535.917,Z 737.114,A -85,B 0,C 180,E1 -2817.559,E2 -2817.559} C_VEL
LIN {X 0,Y 535.933,Z 733.748,A -85,B 0,C 180,E1 -2819.26,E2 -2819.26} C_VEL
LIN {X 0,Y 535.972,Z 728.722,A -85,B 0,C 180,E1 -2820.891,E2 -2820.891} C_VEL
LIN {X 0,Y 536.059,Z 721.789,A -85,B 0,C 180,E1 -2822.533,E2 -2822.533} C_VEL
LIN {X 0,Y 536.202,Z 713.635,A -85,B 0,C 180,E1 -2824.013,E2 -2824.013} C_VEL
LIN {X 0,Y 536.414,Z 703.594,A -85,B 0,C 180,E1 -2825.456,E2 -2825.456} C_VEL
LIN {X 0,Y 536.695,Z 692.234,A -85,B 0,C 180,E1 -2826.765,E2 -2826.765} C_VEL
LIN {X 0,Y 537.025,Z 679.185,A -85,B 0,C 180,E1 -2827.966,E2 -2827.966} C_VEL
LIN {X 0,Y 537.373,Z 665.506,A -85,B 0,C 180,E1 -2828.967,E2 -2828.967} C_VEL
LIN {X 0,Y 537.728,Z 650.25,A -85,B 0,C 180,E1 -2829.83,E2 -2829.83} C_VEL
LIN {X 0,Y 538.04,Z 634.911,A -85,B 0,C 180,E1 -2830.476,E2 -2830.476} C_VEL
LIN {X 0,Y 538.253,Z 618.059,A -85,B 0,C 180,E1 -2830.957,E2 -2830.957} C_VEL
LIN {X 0,Y 538.382,Z 595.599,A -85,B 0,C 180,E1 -2831.307,E2 -2831.307} C_VEL
LIN {X 0,Y 538.715,Z 478.039,A -85,B 0,C 180,E1 -2832.904,E2 -2832.904} C_VEL
LIN {X 0,Y 538.066,Z 472.24,A -85,B 0,C 180,E1 -2833.046,E2 -2833.046} C_VEL
LIN {X 0,Y 538.872,Z 429.115,A -85,B 0,C 180,E1 -2836.414,E2 -2836.414} C_VEL
LIN {X 0,Y 539.475,Z 395.429,A -85,B 0,C 180,E1 -2839.074,E2 -2839.074} C_VEL
LIN {X 0,Y 540.077,Z 355.837,A -85,B 0,C 180,E1 -2842.141,E2 -2842.141} C_VEL
LIN {X 0,Y 540.416,Z 313.922,A -85,B 0,C 180,E1 -2845.388,E2 -2845.388} C_VEL
LIN {X 0,Y 540.347,Z 282.76,A -85,B 0,C 180,E1 -2847.797,E2 -2847.797} C_VEL
LIN {X 0,Y 536.478,Z 269.981,A -85,B 0,C 180,E1 -2849.014,E2 -2849.014} C_VEL
LIN {X 0,Y 536.426,Z 269.667,A -85,B 0,C 180,E1 -2849.784,E2 -2849.784} C_VEL
LIN {X 0,Y 536.424,Z 269.664,A -85,B 0,C 180,E1 -2853.226,E2 -2853.226} C_VEL
LIN {X 0,Y 536.468,Z 269.661,A -85,B 0,C 180,E1 -2856.61,E2 -2856.61} C_VEL
LIN {X 0,Y 536.434,Z 269.664,A -85,B 0,C 180,E1 -2859.946,E2 -2859.946} C_VEL
LIN {X 0,Y 536.423,Z 269.663,A -85,B 0,C 180,E1 -2863.342,E2 -2863.342} C_VEL
LIN {X 0,Y 536.467,Z 269.661,A -85,B 0,C 180,E1 -2866.637,E2 -2866.637} C_VEL
LIN {X 0,Y 536.432,Z 269.664,A -85,B 0,C 180,E1 -2870.017,E2 -2870.017} C_VEL
LIN {X 0,Y 536.425,Z 269.66,A -85,B 0,C 180,E1 -2873.471,E2 -2873.471} C_VEL
LIN {X 0,Y 536.465,Z 269.66,A -85,B 0,C 180,E1 -2876.794,E2 -2876.794} C_VEL
LIN {X 0,Y 536.435,Z 269.664,A -85,B 0,C 180,E1 -2880.106,E2 -2880.106} C_VEL
LIN {X 0,Y 536.429,Z 269.659,A -85,B 0,C 180,E1 -2883.526,E2 -2883.526} C_VEL
LIN {X 0,Y 536.465,Z 269.66,A -85,B 0,C 180,E1 -2886.85,E2 -2886.85} C_VEL
LIN {X 0,Y 536.438,Z 269.662,A -85,B 0,C 180,E1 -2890.232,E2 -2890.232} C_VEL
LIN {X 0,Y 536.427,Z 269.66,A -85,B 0,C 180,E1 -2893.693,E2 -2893.693} C_VEL
LIN {X 0,Y 536.465,Z 269.659,A -85,B 0,C 180,E1 -2897.042,E2 -2897.042} C_VEL
LIN {X 0,Y 536.445,Z 269.664,A -85,B 0,C 180,E1 -2900.398,E2 -2900.398} C_VEL
LIN {X 0,Y 536.43,Z 269.66,A -85,B 0,C 180,E1 -2903.773,E2 -2903.773} C_VEL
LIN {X 0,Y 536.463,Z 269.658,A -85,B 0,C 180,E1 -2907.17,E2 -2907.17} C_VEL
LIN {X 0,Y 536.453,Z 269.663,A -85,B 0,C 180,E1 -2910.585,E2 -2910.585} C_VEL
LIN {X 0,Y 536.429,Z 269.661,A -85,B 0,C 180,E1 -2913.998,E2 -2913.998} C_VEL
LIN {X 0,Y 536.463,Z 269.657,A -85,B 0,C 180,E1 -2917.416,E2 -2917.416} C_VEL
LIN {X 0,Y 536.466,Z 269.664,A -85,B 0,C 180,E1 -2920.858,E2 -2920.858} C_VEL
LIN {X 0,Y 536.431,Z 269.663,A -85,B 0,C 180,E1 -2924.195,E2 -2924.195} C_VEL
LIN {X 0,Y 536.461,Z 269.66,A -85,B 0,C 180,E1 -2927.572,E2 -2927.572} C_VEL
LIN {X 0,Y 536.468,Z 269.663,A -85,B 0,C 180,E1 -2931.004,E2 -2931.004} C_VEL
LIN {X 0,Y 536.428,Z 269.624,A -85,B 0,C 180,E1 -2934.357,E2 -2934.357} C_VEL
LIN {X 0,Y 536.498,Z 269.951,A -85,B 0,C 180,E1 -2934.825,E2 -2934.825} C_VEL
LIN {X 0,Y 543.692,Z 289.122,A -85,B 0,C 180,E1 -2936.798,E2 -2936.798} C_VEL
LIN {X 0,Y 543.017,Z 315.812,A -85,B 0,C 180,E1 -2938.67,E2 -2938.67} C_VEL
LIN {X 0,Y 544.922,Z 328.267,A -85,B 0,C 180,E1 -2938.976,E2 -2938.976} C_VEL
LIN {X 0,Y 543.148,Z 557.81,A -85,B 0,C 180,E1 -2942.278,E2 -2942.278} C_VEL
LIN {X 0,Y 542.802,Z 583.319,A -85,B 0,C 180,E1 -2942.708,E2 -2942.708} C_VEL
LIN {X 0,Y 542.312,Z 604.435,A -85,B 0,C 180,E1 -2943.274,E2 -2943.274} C_VEL
LIN {X 0,Y 541.744,Z 623.594,A -85,B 0,C 180,E1 -2943.978,E2 -2943.978} C_VEL
LIN {X 0,Y 541.035,Z 643.066,A -85,B 0,C 180,E1 -2944.896,E2 -2944.896} C_VEL
LIN {X 0,Y 540.269,Z 661.99,A -85,B 0,C 180,E1 -2946.011,E2 -2946.011} C_VEL
LIN {X 0,Y 539.5,Z 679.409,A -85,B 0,C 180,E1 -2947.25,E2 -2947.25} C_VEL
LIN {X 0,Y 538.724,Z 696.568,A -85,B 0,C 180,E1 -2948.701,E2 -2948.701} C_VEL
LIN {X 0,Y 538.003,Z 712.948,A -85,B 0,C 180,E1 -2950.345,E2 -2950.345} C_VEL
LIN {X 0,Y 537.417,Z 727.069,A -85,B 0,C 180,E1 -2952.012,E2 -2952.012} C_VEL
LIN {X 0,Y 536.939,Z 739.874,A -85,B 0,C 180,E1 -2953.782,E2 -2953.782} C_VEL
LIN {X 0,Y 536.543,Z 751.928,A -85,B 0,C 180,E1 -2955.761,E2 -2955.761} C_VEL
LIN {X 0,Y 536.248,Z 762.399,A -85,B 0,C 180,E1 -2957.838,E2 -2957.838} C_VEL
LIN {X 0,Y 536.08,Z 770.877,A -85,B 0,C 180,E1 -2959.904,E2 -2959.904} C_VEL
LIN {X 0,Y 535.98,Z 777.902,A -85,B 0,C 180,E1 -2962.067,E2 -2962.067} C_VEL
LIN {X 0,Y 535.933,Z 783.144,A -85,B 0,C 180,E1 -2964.219,E2 -2964.219} C_VEL
LIN {X 0,Y 535.908,Z 786.711,A -85,B 0,C 180,E1 -2966.364,E2 -2966.364} C_VEL
LIN {X 0,Y 535.9,Z 788.575,A -85,B 0,C 180,E1 -2968.504,E2 -2968.504} C_VEL
LIN {X 0,Y 535.902,Z 788.873,A -85,B 0,C 180,E1 -2970.643,E2 -2970.643} C_VEL
LIN {X 0,Y 535.911,Z 787.505,A -85,B 0,C 180,E1 -2972.889,E2 -2972.889} C_VEL
LIN {X 0,Y 535.916,Z 784.579,A -85,B 0,C 180,E1 -2975.032,E2 -2975.032} C_VEL
LIN {X 0,Y 535.945,Z 779.971,A -85,B 0,C 180,E1 -2977.182,E2 -2977.182} C_VEL
LIN {X 0,Y 536.019,Z 773.909,A -85,B 0,C 180,E1 -2979.232,E2 -2979.232} C_VEL
LIN {X 0,Y 536.176,Z 765.716,A -85,B 0,C 180,E1 -2981.402,E2 -2981.402} C_VEL
LIN {X 0,Y 536.419,Z 755.985,A -85,B 0,C 180,E1 -2983.474,E2 -2983.474} C_VEL
LIN {X 0,Y 536.765,Z 744.782,A -85,B 0,C 180,E1 -2985.45,E2 -2985.45} C_VEL
LIN {X 0,Y 537.235,Z 732.125,A -85,B 0,C 180,E1 -2987.325,E2 -2987.325} C_VEL
LIN {X 0,Y 537.809,Z 717.951,A -85,B 0,C 180,E1 -2989.1,E2 -2989.1} C_VEL
LIN {X 0,Y 538.49,Z 702.162,A -85,B 0,C 180,E1 -2990.773,E2 -2990.773} C_VEL
LIN {X 0,Y 539.199,Z 685.938,A -85,B 0,C 180,E1 -2992.228,E2 -2992.228} C_VEL
LIN {X 0,Y 539.991,Z 668.119,A -85,B 0,C 180,E1 -2993.576,E2 -2993.576} C_VEL
LIN {X 0,Y 540.789,Z 649.161,A -85,B 0,C 180,E1 -2994.764,E2 -2994.764} C_VEL
LIN {X 0,Y 541.485,Z 630.527,A -85,B 0,C 180,E1 -2995.718,E2 -2995.718} C_VEL
LIN {X 0,Y 542.15,Z 610.603,A -85,B 0,C 180,E1 -2996.524,E2 -2996.524} C_VEL
LIN {X 0,Y 542.707,Z 589.933,A -85,B 0,C 180,E1 -2997.141,E2 -2997.141} C_VEL
LIN {X 0,Y 543.037,Z 569.316,A -85,B 0,C 180,E1 -2997.553,E2 -2997.553} C_VEL
LIN {X 0,Y 544.86,Z 336.081,A -85,B 0,C 180,E1 -3000.91,E2 -3000.91} C_VEL
LIN {X 0,Y 544.695,Z 325.466,A -85,B 0,C 180,E1 -3001.08,E2 -3001.08} C_VEL
LIN {X 0,Y 542.92,Z 315.066,A -85,B 0,C 180,E1 -3001.354,E2 -3001.354} C_VEL
LIN {X 0,Y 543.437,Z 288.327,A -85,B 0,C 180,E1 -3003.223,E2 -3003.223} C_VEL
LIN {X 0,Y 536.523,Z 270.066,A -85,B 0,C 180,E1 -3005.046,E2 -3005.046} C_VEL
LIN {X 0,Y 536.43,Z 269.668,A -85,B 0,C 180,E1 -3005.691,E2 -3005.691} C_VEL
LIN {X 0,Y 536.466,Z 269.664,A -85,B 0,C 180,E1 -3009.048,E2 -3009.048} C_VEL
LIN {X 0,Y 536.46,Z 269.662,A -85,B 0,C 180,E1 -3012.433,E2 -3012.433} C_VEL
LIN {X 0,Y 536.423,Z 269.665,A -85,B 0,C 180,E1 -3015.805,E2 -3015.805} C_VEL
LIN {X 0,Y 536.452,Z 269.666,A -85,B 0,C 180,E1 -3019.176,E2 -3019.176} C_VEL
LIN {X 0,Y 536.464,Z 269.663,A -85,B 0,C 180,E1 -3022.584,E2 -3022.584} C_VEL
LIN {X 0,Y 536.417,Z 269.669,A -85,B 0,C 180,E1 -3025.872,E2 -3025.872} C_VEL
LIN {X 0,Y 536.479,Z 269.923,A -85,B 0,C 180,E1 -3027.247,E2 -3027.247} C_VEL
LIN {X 0,Y 541.851,Z 285.756,A -85,B 0,C 180,E1 -3029.099,E2 -3029.099} C_VEL
LIN {X 0,Y 542.092,Z 288.262,A -85,B 0,C 180,E1 -3029.337,E2 -3029.337} C_VEL
LIN {X 0,Y 540.798,Z 330.21,A -85,B 0,C 180,E1 -3032.787,E2 -3032.787} C_VEL
LIN {X 0,Y 540.524,Z 342.365,A -85,B 0,C 180,E1 -3033.748,E2 -3033.748} C_VEL
LIN {X 0,Y 542.297,Z 354.174,A -85,B 0,C 180,E1 -3034.024,E2 -3034.024} C_VEL
LIN {X 0,Y 540.93,Z 559.878,A -85,B 0,C 180,E1 -3036.926,E2 -3036.926} C_VEL
LIN {X 0,Y 540.561,Z 579.589,A -85,B 0,C 180,E1 -3037.409,E2 -3037.409} C_VEL
LIN {X 0,Y 540.109,Z 597.611,A -85,B 0,C 180,E1 -3038.043,E2 -3038.043} C_VEL
LIN {X 0,Y 539.561,Z 615.488,A -85,B 0,C 180,E1 -3038.874,E2 -3038.874} C_VEL
LIN {X 0,Y 538.941,Z 633.351,A -85,B 0,C 180,E1 -3039.927,E2 -3039.927} C_VEL
LIN {X 0,Y 538.339,Z 650.126,A -85,B 0,C 180,E1 -3041.146,E2 -3041.146} C_VEL
LIN {X 0,Y 537.743,Z 665.732,A -85,B 0,C 180,E1 -3042.527,E2 -3042.527} C_VEL
LIN {X 0,Y 537.229,Z 679.731,A -85,B 0,C 180,E1 -3044.012,E2 -3044.012} C_VEL
LIN {X 0,Y 536.794,Z 692.735,A -85,B 0,C 180,E1 -3045.657,E2 -3045.657} C_VEL
LIN {X 0,Y 536.451,Z 704.2,A -85,B 0,C 180,E1 -3047.405,E2 -3047.405} C_VEL
LIN {X 0,Y 536.197,Z 714.521,A -85,B 0,C 180,E1 -3049.332,E2 -3049.332} C_VEL
LIN {X 0,Y 536.044,Z 722.975,A -85,B 0,C 180,E1 -3051.311,E2 -3051.311} C_VEL
LIN {X 0,Y 535.953,Z 729.726,A -85,B 0,C 180,E1 -3053.358,E2 -3053.358} C_VEL
LIN {X 0,Y 535.92,Z 734.557,A -85,B 0,C 180,E1 -3055.399,E2 -3055.399} C_VEL
LIN {X 0,Y 535.913,Z 737.584,A -85,B 0,C 180,E1 -3057.434,E2 -3057.434} C_VEL
LIN {X 0,Y 535.909,Z 738.883,A -85,B 0,C 180,E1 -3059.466,E2 -3059.466} C_VEL
LIN {X 0,Y 535.911,Z 738.47,A -85,B 0,C 180,E1 -3061.604,E2 -3061.604} C_VEL
LIN {X 0,Y 535.909,Z 736.343,A -85,B 0,C 180,E1 -3063.637,E2 -3063.637} C_VEL
LIN {X 0,Y 535.936,Z 732.458,A -85,B 0,C 180,E1 -3065.675,E2 -3065.675} C_VEL
LIN {X 0,Y 535.986,Z 726.718,A -85,B 0,C 180,E1 -3067.719,E2 -3067.719} C_VEL
LIN {X 0,Y 536.111,Z 718.986,A -85,B 0,C 180,E1 -3069.772,E2 -3069.772} C_VEL
LIN {X 0,Y 536.314,Z 709.616,A -85,B 0,C 180,E1 -3071.725,E2 -3071.725} C_VEL
LIN {X 0,Y 536.612,Z 698.614,A -85,B 0,C 180,E1 -3073.579,E2 -3073.579} C_VEL
LIN {X 0,Y 537.018,Z 685.955,A -85,B 0,C 180,E1 -3075.331,E2 -3075.331} C_VEL
LIN {X 0,Y 537.514,Z 672.061,A -85,B 0,C 180,E1 -3076.925,E2 -3076.925} C_VEL
LIN {X 0,Y 538.075,Z 657.098,A -85,B 0,C 180,E1 -3078.359,E2 -3078.359} C_VEL
LIN {X 0,Y 538.673,Z 641.059,A -85,B 0,C 180,E1 -3079.632,E2 -3079.632} C_VEL
LIN {X 0,Y 539.277,Z 624.057,A -85,B 0,C 180,E1 -3080.741,E2 -3080.741} C_VEL
LIN {X 0,Y 539.834,Z 607.194,A -85,B 0,C 180,E1 -3081.629,E2 -3081.629} C_VEL
LIN {X 0,Y 540.353,Z 588.542,A -85,B 0,C 180,E1 -3082.389,E2 -3082.389} C_VEL
LIN {X 0,Y 540.775,Z 568.878,A -85,B 0,C 180,E1 -3082.97,E2 -3082.97} C_VEL
LIN {X 0,Y 541.052,Z 549.078,A -85,B 0,C 180,E1 -3083.341,E2 -3083.341} C_VEL
LIN {X 0,Y 541.182,Z 527.864,A -85,B 0,C 180,E1 -3083.636,E2 -3083.636} C_VEL
LIN {X 0,Y 540.307,Z 520.275,A -85,B 0,C 180,E1 -3083.784,E2 -3083.784} C_VEL
LIN {X 0,Y 534.727,Z 500.431,A -85,B 0,C 180,E1 -3084.334,E2 -3084.334} C_VEL
LIN {X 0,Y 534.074,Z 493.908,A -85,B 0,C 180,E1 -3084.46,E2 -3084.46} C_VEL
LIN {X 0,Y 534.906,Z 352.739,A -85,B 0,C 180,E1 -3086.475,E2 -3086.475} C_VEL
LIN {X 0,Y 533.102,Z 342.045,A -85,B 0,C 180,E1 -3086.753,E2 -3086.753} C_VEL
LIN {X 0,Y 534.497,Z 300.157,A -85,B 0,C 180,E1 -3090.213,E2 -3090.213} C_VEL
LIN {X 0,Y 534.882,Z 289.528,A -85,B 0,C 180,E1 -3091.113,E2 -3091.113} C_VEL
LIN {X 0,Y 528.554,Z 270.846,A -85,B 0,C 180,E1 -3093.254,E2 -3093.254} C_VEL
LIN {X 0,Y 528.493,Z 270.654,A -85,B 0,C 180,E1 -3096.48,E2 -3096.48} C_VEL
LIN {X 0,Y 528.494,Z 270.65,A -85,B 0,C 180,E1 -3099.983,E2 -3099.983} C_VEL
LIN {X 0,Y 528.526,Z 270.647,A -85,B 0,C 180,E1 -3103.41,E2 -3103.41} C_VEL
LIN {X 0,Y 528.52,Z 270.65,A -85,B 0,C 180,E1 -3106.925,E2 -3106.925} C_VEL
LIN {X 0,Y 528.516,Z 270.653,A -85,B 0,C 180,E1 -3110.352,E2 -3110.352} C_VEL
LIN {X 0,Y 528.516,Z 270.647,A -85,B 0,C 180,E1 -3113.883,E2 -3113.883} C_VEL
LIN {X 0,Y 528.507,Z 270.648,A -85,B 0,C 180,E1 -3117.243,E2 -3117.243} C_VEL
LIN {X 0,Y 528.503,Z 270.647,A -85,B 0,C 180,E1 -3120.783,E2 -3120.783} C_VEL
LIN {X 0,Y 528.526,Z 270.648,A -85,B 0,C 180,E1 -3124.224,E2 -3124.224} C_VEL
LIN {X 0,Y 528.519,Z 270.649,A -85,B 0,C 180,E1 -3127.684,E2 -3127.684} C_VEL
LIN {X 0,Y 528.476,Z 270.652,A -85,B 0,C 180,E1 -3131.084,E2 -3131.084} C_VEL
LIN {X 0,Y 528.481,Z 270.646,A -85,B 0,C 180,E1 -3134.527,E2 -3134.527} C_VEL
LIN {X 0,Y 528.509,Z 270.651,A -85,B 0,C 180,E1 -3137.766,E2 -3137.766} C_VEL
LIN {X 0,Y 528.497,Z 270.87,A -85,B 0,C 180,E1 -3140.47,E2 -3140.47} C_VEL
LIN {X 0,Y 533.456,Z 286.886,A -85,B 0,C 180,E1 -3142.081,E2 -3142.081} C_VEL
LIN {X 0,Y 533.075,Z 326.99,A -85,B 0,C 180,E1 -3145.265,E2 -3145.265} C_VEL
LIN {X 0,Y 532.459,Z 368.362,A -85,B 0,C 180,E1 -3148.546,E2 -3148.546} C_VEL
LIN {X 0,Y 531.647,Z 411.901,A -85,B 0,C 180,E1 -3151.993,E2 -3151.993} C_VEL
LIN {X 0,Y 530.729,Z 455.611,A -85,B 0,C 180,E1 -3155.458,E2 -3155.458} C_VEL
LIN {X 0,Y 530.457,Z 473.352,A -85,B 0,C 180,E1 -3156.822,E2 -3156.822} C_VEL
LIN {X 0,Y 531.307,Z 482.893,A -85,B 0,C 180,E1 -3156.994,E2 -3156.994} C_VEL
LIN {X 0,Y 530.599,Z 615.85,A -85,B 0,C 180,E1 -3158.847,E2 -3158.847} C_VEL
LIN {X 0,Y 530.385,Z 631.772,A -85,B 0,C 180,E1 -3159.267,E2 -3159.267} C_VEL
LIN {X 0,Y 530.074,Z 647.293,A -85,B 0,C 180,E1 -3159.882,E2 -3159.882} C_VEL
LIN {X 0,Y 529.71,Z 661.751,A -85,B 0,C 180,E1 -3160.659,E2 -3160.659} C_VEL
LIN {X 0,Y 529.286,Z 676.065,A -85,B 0,C 180,E1 -3161.66,E2 -3161.66} C_VEL
LIN {X 0,Y 528.924,Z 688.726,A -85,B 0,C 180,E1 -3162.777,E2 -3162.777} C_VEL
LIN {X 0,Y 528.567,Z 700.857,A -85,B 0,C 180,E1 -3164.123,E2 -3164.123} C_VEL
LIN {X 0,Y 528.292,Z 711.425,A -85,B 0,C 180,E1 -3165.589,E2 -3165.589} C_VEL
LIN {X 0,Y 528.102,Z 720.477,A -85,B 0,C 180,E1 -3167.177,E2 -3167.177} C_VEL
LIN {X 0,Y 527.995,Z 727.509,A -85,B 0,C 180,E1 -3168.778,E2 -3168.778} C_VEL
LIN {X 0,Y 527.936,Z 733.064,A -85,B 0,C 180,E1 -3170.509,E2 -3170.509} C_VEL
LIN {X 0,Y 527.923,Z 736.631,A -85,B 0,C 180,E1 -3172.158,E2 -3172.158} C_VEL
LIN {X 0,Y 527.916,Z 738.604,A -85,B 0,C 180,E1 -3173.909,E2 -3173.909} C_VEL
LIN {X 0,Y 527.915,Z 738.87,A -85,B 0,C 180,E1 -3175.702,E2 -3175.702} C_VEL
LIN {X 0,Y 527.917,Z 737.398,A -85,B 0,C 180,E1 -3177.401,E2 -3177.401} C_VEL
LIN {X 0,Y 527.935,Z 733.922,A -85,B 0,C 180,E1 -3179.249,E2 -3179.249} C_VEL
LIN {X 0,Y 527.978,Z 728.938,A -85,B 0,C 180,E1 -3180.921,E2 -3180.921} C_VEL
LIN {X 0,Y 528.083,Z 721.748,A -85,B 0,C 180,E1 -3182.655,E2 -3182.655} C_VEL
LIN {X 0,Y 528.251,Z 713.297,A -85,B 0,C 180,E1 -3184.203,E2 -3184.203} C_VEL
LIN {X 0,Y 528.524,Z 702.456,A -85,B 0,C 180,E1 -3185.77,E2 -3185.77} C_VEL
LIN {X 0,Y 528.854,Z 690.914,A -85,B 0,C 180,E1 -3187.091,E2 -3187.091} C_VEL
LIN {X 0,Y 529.242,Z 677.872,A -85,B 0,C 180,E1 -3188.29,E2 -3188.29} C_VEL
LIN {X 0,Y 529.638,Z 664.081,A -85,B 0,C 180,E1 -3189.284,E2 -3189.284} C_VEL
LIN {X 0,Y 530.042,Z 648.995,A -85,B 0,C 180,E1 -3190.131,E2 -3190.131} C_VEL
LIN {X 0,Y 530.364,Z 632.881,A -85,B 0,C 180,E1 -3190.786,E2 -3190.786} C_VEL
LIN {X 0,Y 530.581,Z 616.78,A -85,B 0,C 180,E1 -3191.227,E2 -3191.227} C_VEL
LIN {X 0,Y 530.833,Z 568.061,A -85,B 0,C 180,E1 -3191.928,E2 -3191.928} C_VEL
LIN {X 0,Y 531.109,Z 478.885,A -85,B 0,C 180,E1 -3193.159,E2 -3193.159} C_VEL
LIN {X 0,Y 530.394,Z 472.628,A -85,B 0,C 180,E1 -3193.309,E2 -3193.309} C_VEL
LIN {X 0,Y 531.251,Z 429.763,A -85,B 0,C 180,E1 -3196.684,E2 -3196.684} C_VEL
LIN {X 0,Y 532.007,Z 389.605,A -85,B 0,C 180,E1 -3199.861,E2 -3199.861} C_VEL
LIN {X 0,Y 532.616,Z 350.06,A -85,B 0,C 180,E1 -3202.943,E2 -3202.943} C_VEL
LIN {X 0,Y 532.94,Z 312.405,A -85,B 0,C 180,E1 -3205.877,E2 -3205.877} C_VEL
LIN {X 0,Y 532.852,Z 285.087,A -85,B 0,C 180,E1 -3208.007,E2 -3208.007} C_VEL
LIN {X 0,Y 528.518,Z 270.929,A -85,B 0,C 180,E1 -3209.377,E2 -3209.377} C_VEL
LIN {X 0,Y 528.488,Z 270.655,A -85,B 0,C 180,E1 -3211.771,E2 -3211.771} C_VEL
LIN {X 0,Y 528.484,Z 270.653,A -85,B 0,C 180,E1 -3215.284,E2 -3215.284} C_VEL
LIN {X 0,Y 528.528,Z 270.648,A -85,B 0,C 180,E1 -3218.585,E2 -3218.585} C_VEL
LIN {X 0,Y 528.492,Z 270.65,A -85,B 0,C 180,E1 -3221.924,E2 -3221.924} C_VEL
LIN {X 0,Y 528.488,Z 270.649,A -85,B 0,C 180,E1 -3225.314,E2 -3225.314} C_VEL
LIN {X 0,Y 528.527,Z 270.65,A -85,B 0,C 180,E1 -3228.653,E2 -3228.653} C_VEL
LIN {X 0,Y 528.496,Z 270.652,A -85,B 0,C 180,E1 -3232.061,E2 -3232.061} C_VEL
LIN {X 0,Y 528.488,Z 270.649,A -85,B 0,C 180,E1 -3235.442,E2 -3235.442} C_VEL
LIN {X 0,Y 528.527,Z 270.649,A -85,B 0,C 180,E1 -3238.807,E2 -3238.807} C_VEL
LIN {X 0,Y 528.499,Z 270.652,A -85,B 0,C 180,E1 -3242.168,E2 -3242.168} C_VEL
LIN {X 0,Y 528.486,Z 270.65,A -85,B 0,C 180,E1 -3245.646,E2 -3245.646} C_VEL
LIN {X 0,Y 528.527,Z 270.646,A -85,B 0,C 180,E1 -3248.924,E2 -3248.924} C_VEL
LIN {X 0,Y 528.506,Z 270.653,A -85,B 0,C 180,E1 -3252.344,E2 -3252.344} C_VEL
LIN {X 0,Y 528.49,Z 270.647,A -85,B 0,C 180,E1 -3255.696,E2 -3255.696} C_VEL
LIN {X 0,Y 528.526,Z 270.647,A -85,B 0,C 180,E1 -3259.103,E2 -3259.103} C_VEL
LIN {X 0,Y 528.519,Z 270.651,A -85,B 0,C 180,E1 -3262.584,E2 -3262.584} C_VEL
LIN {X 0,Y 528.489,Z 270.651,A -85,B 0,C 180,E1 -3266.022,E2 -3266.022} C_VEL
LIN {X 0,Y 528.514,Z 270.645,A -85,B 0,C 180,E1 -3269.464,E2 -3269.464} C_VEL
LIN {X 0,Y 528.526,Z 270.652,A -85,B 0,C 180,E1 -3272.884,E2 -3272.884} C_VEL
LIN {X 0,Y 528.494,Z 270.652,A -85,B 0,C 180,E1 -3276.31,E2 -3276.31} C_VEL
LIN {X 0,Y 528.5,Z 270.648,A -85,B 0,C 180,E1 -3279.819,E2 -3279.819} C_VEL
LIN {X 0,Y 528.526,Z 270.651,A -85,B 0,C 180,E1 -3283.222,E2 -3283.222} C_VEL
LIN {X 0,Y 528.509,Z 270.654,A -85,B 0,C 180,E1 -3286.63,E2 -3286.63} C_VEL
LIN {X 0,Y 528.496,Z 270.651,A -85,B 0,C 180,E1 -3290.015,E2 -3290.015} C_VEL
LIN {X 0,Y 528.519,Z 270.616,A -85,B 0,C 180,E1 -3293.333,E2 -3293.333} C_VEL
LIN {X 0,Y 528.529,Z 270.894,A -85,B 0,C 180,E1 -3294.297,E2 -3294.297} C_VEL
LIN {X 0,Y 530.564,Z 276.356,A -85,B 0,C 180,E1 -3294.918,E2 -3294.918} C_VEL
LIN {X 0,Y 536.57,Z 291.928,A -85,B 0,C 180,E1 -3296.527,E2 -3296.527} C_VEL
LIN {X 0,Y 535.869,Z 316.027,A -85,B 0,C 180,E1 -3298.239,E2 -3298.239} C_VEL
LIN {X 0,Y 537.956,Z 329.446,A -85,B 0,C 180,E1 -3298.572,E2 -3298.572} C_VEL
LIN {X 0,Y 536.141,Z 549.123,A -85,B 0,C 180,E1 -3301.754,E2 -3301.754} C_VEL
LIN {X 0,Y 535.77,Z 580.397,A -85,B 0,C 180,E1 -3302.251,E2 -3302.251} C_VEL
LIN {X 0,Y 535.266,Z 600.963,A -85,B 0,C 180,E1 -3302.774,E2 -3302.774} C_VEL
LIN {X 0,Y 534.596,Z 620.781,A -85,B 0,C 180,E1 -3303.48,E2 -3303.48} C_VEL
LIN {X 0,Y 533.837,Z 639.893,A -85,B 0,C 180,E1 -3304.366,E2 -3304.366} C_VEL
LIN {X 0,Y 532.985,Z 658.752,A -85,B 0,C 180,E1 -3305.449,E2 -3305.449} C_VEL
LIN {X 0,Y 532.069,Z 677.587,A -85,B 0,C 180,E1 -3306.769,E2 -3306.769} C_VEL
LIN {X 0,Y 531.234,Z 694.408,A -85,B 0,C 180,E1 -3308.18,E2 -3308.18} C_VEL
LIN {X 0,Y 530.443,Z 710.413,A -85,B 0,C 180,E1 -3309.766,E2 -3309.766} C_VEL
LIN {X 0,Y 529.729,Z 725.368,A -85,B 0,C 180,E1 -3311.514,E2 -3311.514} C_VEL
LIN {X 0,Y 529.125,Z 739.131,A -85,B 0,C 180,E1 -3313.423,E2 -3313.423} C_VEL
LIN {X 0,Y 528.68,Z 750.657,A -85,B 0,C 180,E1 -3315.321,E2 -3315.321} C_VEL
LIN {X 0,Y 528.348,Z 760.855,A -85,B 0,C 180,E1 -3317.32,E2 -3317.32} C_VEL
LIN {X 0,Y 528.124,Z 770.067,A -85,B 0,C 180,E1 -3319.53,E2 -3319.53} C_VEL
LIN {X 0,Y 528.002,Z 777.295,A -85,B 0,C 180,E1 -3321.727,E2 -3321.727} C_VEL
LIN {X 0,Y 527.944,Z 782.73,A -85,B 0,C 180,E1 -3323.913,E2 -3323.913} C_VEL
LIN {X 0,Y 527.918,Z 786.404,A -85,B 0,C 180,E1 -3326.092,E2 -3326.092} C_VEL
LIN {X 0,Y 527.906,Z 788.443,A -85,B 0,C 180,E1 -3328.265,E2 -3328.265} C_VEL
LIN {X 0,Y 527.9,Z 788.895,A -85,B 0,C 180,E1 -3330.544,E2 -3330.544} C_VEL
LIN {X 0,Y 527.911,Z 787.729,A -85,B 0,C 180,E1 -3332.715,E2 -3332.715} C_VEL
LIN {X 0,Y 527.922,Z 784.968,A -85,B 0,C 180,E1 -3334.89,E2 -3334.89} C_VEL
LIN {X 0,Y 527.948,Z 780.464,A -85,B 0,C 180,E1 -3337.079,E2 -3337.079} C_VEL
LIN {X 0,Y 528.031,Z 774.263,A -85,B 0,C 180,E1 -3339.263,E2 -3339.263} C_VEL
LIN {X 0,Y 528.207,Z 766.173,A -85,B 0,C 180,E1 -3341.465,E2 -3341.465} C_VEL
LIN {X 0,Y 528.478,Z 756.557,A -85,B 0,C 180,E1 -3343.569,E2 -3343.569} C_VEL
LIN {X 0,Y 528.869,Z 745.481,A -85,B 0,C 180,E1 -3345.574,E2 -3345.574} C_VEL
LIN {X 0,Y 529.395,Z 732.863,A -85,B 0,C 180,E1 -3347.488,E2 -3347.488} C_VEL
LIN {X 0,Y 530.029,Z 718.878,A -85,B 0,C 180,E1 -3349.277,E2 -3349.277} C_VEL
LIN {X 0,Y 530.753,Z 703.881,A -85,B 0,C 180,E1 -3350.911,E2 -3350.911} C_VEL
LIN {X 0,Y 531.581,Z 687.27,A -85,B 0,C 180,E1 -3352.448,E2 -3352.448} C_VEL
LIN {X 0,Y 532.465,Z 669.74,A -85,B 0,C 180,E1 -3353.812,E2 -3353.812} C_VEL
LIN {X 0,Y 533.347,Z 651.268,A -85,B 0,C 180,E1 -3355.009,E2 -3355.009} C_VEL
LIN {X 0,Y 534.152,Z 632.343,A -85,B 0,C 180,E1 -3356.013,E2 -3356.013} C_VEL
LIN {X 0,Y 534.891,Z 612.583,A -85,B 0,C 180,E1 -3356.836,E2 -3356.836} C_VEL
LIN {X 0,Y 535.481,Z 592.698,A -85,B 0,C 180,E1 -3357.458,E2 -3357.458} C_VEL
LIN {X 0,Y 535.906,Z 571.719,A -85,B 0,C 180,E1 -3357.909,E2 -3357.909} C_VEL
LIN {X 0,Y 537.478,Z 381.035,A -85,B 0,C 180,E1 -3360.663,E2 -3360.663} C_VEL
LIN {X 0,Y 537.602,Z 326.941,A -85,B 0,C 180,E1 -3361.445,E2 -3361.445} C_VEL
LIN {X 0,Y 535.65,Z 315.573,A -85,B 0,C 180,E1 -3361.734,E2 -3361.734} C_VEL
LIN {X 0,Y 536.239,Z 291.369,A -85,B 0,C 180,E1 -3363.447,E2 -3363.447} C_VEL
LIN {X 0,Y 528.555,Z 271.061,A -85,B 0,C 180,E1 -3365.536,E2 -3365.536} C_VEL
LIN {X 0,Y 528.509,Z 270.655,A -85,B 0,C 180,E1 -3366.176,E2 -3366.176} C_VEL
LIN {X 0,Y 528.489,Z 270.655,A -85,B 0,C 180,E1 -3369.646,E2 -3369.646} C_VEL
LIN {X 0,Y 528.525,Z 270.653,A -85,B 0,C 180,E1 -3372.936,E2 -3372.936} C_VEL
LIN {X 0,Y 528.508,Z 270.652,A -85,B 0,C 180,E1 -3376.329,E2 -3376.329} C_VEL
LIN {X 0,Y 528.483,Z 270.656,A -85,B 0,C 180,E1 -3379.682,E2 -3379.682} C_VEL
LIN {X 0,Y 528.522,Z 270.654,A -85,B 0,C 180,E1 -3383.016,E2 -3383.016} C_VEL
LIN {X 0,Y 528.499,Z 270.655,A -85,B 0,C 180,E1 -3386.35,E2 -3386.35} C_VEL
LIN {X 0,Y 528.597,Z 271.112,A -85,B 0,C 180,E1 -3386.744,E2 -3386.744} C_VEL
LIN {X 0,Y 534.257,Z 287.303,A -85,B 0,C 180,E1 -3388.687,E2 -3388.687} C_VEL
LIN {X 0,Y 534.992,Z 290.3,A -85,B 0,C 180,E1 -3389.01,E2 -3389.01} C_VEL
LIN {X 0,Y 533.49,Z 329.28,A -85,B 0,C 180,E1 -3392.303,E2 -3392.303} C_VEL
LIN {X 0,Y 533.154,Z 342.603,A -85,B 0,C 180,E1 -3393.362,E2 -3393.362} C_VEL
LIN {X 0,Y 535.101,Z 355.243,A -85,B 0,C 180,E1 -3393.663,E2 -3393.663} C_VEL
LIN {X 0,Y 533.574,Z 559.734,A -85,B 0,C 180,E1 -3396.586,E2 -3396.586} C_VEL
LIN {X 0,Y 533.162,Z 579.368,A -85,B 0,C 180,E1 -3397.071,E2 -3397.071} C_VEL
LIN {X 0,Y 532.643,Z 598.047,A -85,B 0,C 180,E1 -3397.736,E2 -3397.736} C_VEL
LIN {X 0,Y 532.045,Z 615.497,A -85,B 0,C 180,E1 -3398.561,E2 -3398.561} C_VEL
LIN {X 0,Y 531.351,Z 633.357,A -85,B 0,C 180,E1 -3399.628,E2 -3399.628} C_VEL
LIN {X 0,Y 530.673,Z 650.135,A -85,B 0,C 180,E1 -3400.863,E2 -3400.863} C_VEL
LIN {X 0,Y 530.001,Z 665.776,A -85,B 0,C 180,E1 -3402.268,E2 -3402.268} C_VEL
LIN {X 0,Y 529.424,Z 679.736,A -85,B 0,C 180,E1 -3403.769,E2 -3403.769} C_VEL
LIN {X 0,Y 528.923,Z 692.743,A -85,B 0,C 180,E1 -3405.439,E2 -3405.439} C_VEL
LIN {X 0,Y 528.529,Z 704.205,A -85,B 0,C 180,E1 -3407.213,E2 -3407.213} C_VEL
LIN {X 0,Y 528.25,Z 714.139,A -85,B 0,C 180,E1 -3409.09,E2 -3409.09} C_VEL
LIN {X 0,Y 528.07,Z 722.57,A -85,B 0,C 180,E1 -3411.068,E2 -3411.068} C_VEL
LIN {X 0,Y 527.969,Z 729.125,A -85,B 0,C 180,E1 -3413.039,E2 -3413.039} C_VEL
LIN {X 0,Y 527.932,Z 734.152,A -85,B 0,C 180,E1 -3415.111,E2 -3415.111} C_VEL
LIN {X 0,Y 527.912,Z 737.34,A -85,B 0,C 180,E1 -3417.178,E2 -3417.178} C_VEL
LIN {X 0,Y 527.917,Z 738.83,A -85,B 0,C 180,E1 -3419.241,E2 -3419.241} C_VEL
LIN {X 0,Y 527.911,Z 738.671,A -85,B 0,C 180,E1 -3421.303,E2 -3421.303} C_VEL
LIN {X 0,Y 527.915,Z 736.802,A -85,B 0,C 180,E1 -3423.366,E2 -3423.366} C_VEL
LIN {X 0,Y 527.932,Z 733.178,A -85,B 0,C 180,E1 -3425.434,E2 -3425.434} C_VEL
LIN {X 0,Y 527.986,Z 727.754,A -85,B 0,C 180,E1 -3427.509,E2 -3427.509} C_VEL
LIN {X 0,Y 528.113,Z 720.829,A -85,B 0,C 180,E1 -3429.481,E2 -3429.481} C_VEL
LIN {X 0,Y 528.317,Z 711.915,A -85,B 0,C 180,E1 -3431.462,E2 -3431.462} C_VEL
LIN {X 0,Y 528.625,Z 701.393,A -85,B 0,C 180,E1 -3433.342,E2 -3433.342} C_VEL
LIN {X 0,Y 529.045,Z 689.306,A -85,B 0,C 180,E1 -3435.119,E2 -3435.119} C_VEL
LIN {X 0,Y 529.58,Z 675.608,A -85,B 0,C 180,E1 -3436.791,E2 -3436.791} C_VEL
LIN {X 0,Y 530.18,Z 661.357,A -85,B 0,C 180,E1 -3438.244,E2 -3438.244} C_VEL
LIN {X 0,Y 530.858,Z 645.547,A -85,B 0,C 180,E1 -3439.589,E2 -3439.589} C_VEL
LIN {X 0,Y 531.552,Z 628.56,A -85,B 0,C 180,E1 -3440.773,E2 -3440.773} C_VEL
LIN {X 0,Y 532.227,Z 610.564,A -85,B 0,C 180,E1 -3441.78,E2 -3441.78} C_VEL
LIN {X 0,Y 532.834,Z 591.907,A -85,B 0,C 180,E1 -3442.595,E2 -3442.595} C_VEL
LIN {X 0,Y 533.31,Z 572.811,A -85,B 0,C 180,E1 -3443.206,E2 -3443.206} C_VEL
LIN {X 0,Y 533.655,Z 552.956,A -85,B 0,C 180,E1 -3443.621,E2 -3443.621} C_VEL
LIN {X 0,Y 534.074,Z 493.908,A -85,B 0,C 180,E1 -3444.46,E2 -3444.46} C_VEL
LIN {X 0,Y 533.205,Z 486.322,A -85,B 0,C 180,E1 -3444.612,E2 -3444.612} C_VEL
LIN {X 0,Y 527.673,Z 466.49,A -85,B 0,C 180,E1 -3445.179,E2 -3445.179} C_VEL
LIN {X 0,Y 527.04,Z 459.968,A -85,B 0,C 180,E1 -3445.307,E2 -3445.307} C_VEL
LIN {X 0,Y 527.743,Z 353.96,A -85,B 0,C 180,E1 -3446.844,E2 -3446.844} C_VEL
LIN {X 0,Y 525.72,Z 341.772,A -85,B 0,C 180,E1 -3447.174,E2 -3447.174} C_VEL
LIN {X 0,Y 527.445,Z 297.433,A -85,B 0,C 180,E1 -3450.913,E2 -3450.913} C_VEL
LIN {X 0,Y 527.649,Z 292.421,A -85,B 0,C 180,E1 -3451.343,E2 -3451.343} C_VEL
LIN {X 0,Y 520.596,Z 271.913,A -85,B 0,C 180,E1 -3453.733,E2 -3453.733} C_VEL
LIN {X 0,Y 520.577,Z 271.605,A -85,B 0,C 180,E1 -3454.916,E2 -3454.916} C_VEL
LIN {X 0,Y 520.553,Z 271.642,A -85,B 0,C 180,E1 -3458.346,E2 -3458.346} C_VEL
LIN {X 0,Y 520.564,Z 271.635,A -85,B 0,C 180,E1 -3461.819,E2 -3461.819} C_VEL
LIN {X 0,Y 520.584,Z 271.639,A -85,B 0,C 180,E1 -3465.179,E2 -3465.179} C_VEL
LIN {X 0,Y 520.589,Z 271.641,A -85,B 0,C 180,E1 -3468.675,E2 -3468.675} C_VEL
LIN {X 0,Y 520.573,Z 271.64,A -85,B 0,C 180,E1 -3472.131,E2 -3472.131} C_VEL
LIN {X 0,Y 520.583,Z 271.634,A -85,B 0,C 180,E1 -3475.62,E2 -3475.62} C_VEL
LIN {X 0,Y 520.561,Z 271.637,A -85,B 0,C 180,E1 -3479.018,E2 -3479.018} C_VEL
LIN {X 0,Y 520.58,Z 271.642,A -85,B 0,C 180,E1 -3482.426,E2 -3482.426} C_VEL
LIN {X 0,Y 520.586,Z 271.632,A -85,B 0,C 180,E1 -3485.851,E2 -3485.851} C_VEL
LIN {X 0,Y 520.544,Z 271.638,A -85,B 0,C 180,E1 -3489.184,E2 -3489.184} C_VEL
LIN {X 0,Y 520.541,Z 271.645,A -85,B 0,C 180,E1 -3492.679,E2 -3492.679} C_VEL
LIN {X 0,Y 520.584,Z 271.616,A -85,B 0,C 180,E1 -3495.994,E2 -3495.994} C_VEL
LIN {X 0,Y 520.528,Z 271.626,A -85,B 0,C 180,E1 -3499.373,E2 -3499.373} C_VEL
LIN {X 0,Y 520.604,Z 271.906,A -85,B 0,C 180,E1 -3500.091,E2 -3500.091} C_VEL
LIN {X 0,Y 526.056,Z 289.295,A -85,B 0,C 180,E1 -3501.858,E2 -3501.858} C_VEL
LIN {X 0,Y 525.617,Z 328.259,A -85,B 0,C 180,E1 -3504.979,E2 -3504.979} C_VEL
LIN {X 0,Y 524.934,Z 369.946,A -85,B 0,C 180,E1 -3508.307,E2 -3508.307} C_VEL
LIN {X 0,Y 524.037,Z 413.741,A -85,B 0,C 180,E1 -3511.803,E2 -3511.803} C_VEL
LIN {X 0,Y 523.081,Z 456.223,A -85,B 0,C 180,E1 -3515.196,E2 -3515.196} C_VEL
LIN {X 0,Y 522.811,Z 473.835,A -85,B 0,C 180,E1 -3516.553,E2 -3516.553} C_VEL
LIN {X 0,Y 523.704,Z 483.653,A -85,B 0,C 180,E1 -3516.731,E2 -3516.731} C_VEL
LIN {X 0,Y 522.921,Z 616.085,A -85,B 0,C 180,E1 -3518.604,E2 -3518.604} C_VEL
LIN {X 0,Y 522.693,Z 631.969,A -85,B 0,C 180,E1 -3519.027,E2 -3519.027} C_VEL
LIN {X 0,Y 522.333,Z 648.53,A -85,B 0,C 180,E1 -3519.696,E2 -3519.696} C_VEL
LIN {X 0,Y 521.931,Z 662.754,A -85,B 0,C 180,E1 -3520.484,E2 -3520.484} C_VEL
LIN {X 0,Y 521.46,Z 677.361,A -85,B 0,C 180,E1 -3521.532,E2 -3521.532} C_VEL
LIN {X 0,Y 521.044,Z 690.15,A -85,B 0,C 180,E1 -3522.701,E2 -3522.701} C_VEL
LIN {X 0,Y 520.675,Z 701.58,A -85,B 0,C 180,E1 -3524.001,E2 -3524.001} C_VEL
LIN {X 0,Y 520.383,Z 711.333,A -85,B 0,C 180,E1 -3525.375,E2 -3525.375} C_VEL
LIN {X 0,Y 520.152,Z 720.372,A -85,B 0,C 180,E1 -3526.987,E2 -3526.987} C_VEL
LIN {X 0,Y 520.018,Z 727.428,A -85,B 0,C 180,E1 -3528.611,E2 -3528.611} C_VEL
LIN {X 0,Y 519.946,Z 732.976,A -85,B 0,C 180,E1 -3530.367,E2 -3530.367} C_VEL
LIN {X 0,Y 519.924,Z 736.732,A -85,B 0,C 180,E1 -3532.142,E2 -3532.142} C_VEL
LIN {X 0,Y 519.917,Z 738.705,A -85,B 0,C 180,E1 -3534.008,E2 -3534.008} C_VEL
LIN {X 0,Y 519.916,Z 738.85,A -85,B 0,C 180,E1 -3535.838,E2 -3535.838} C_VEL
LIN {X 0,Y 519.919,Z 737.028,A -85,B 0,C 180,E1 -3537.734,E2 -3537.734} C_VEL
LIN {X 0,Y 519.941,Z 733.601,A -85,B 0,C 180,E1 -3539.49,E2 -3539.49} C_VEL
LIN {X 0,Y 520.007,Z 728.163,A -85,B 0,C 180,E1 -3541.273,E2 -3541.273} C_VEL
LIN {X 0,Y 520.139,Z 721.127,A -85,B 0,C 180,E1 -3542.955,E2 -3542.955} C_VEL
LIN {X 0,Y 520.364,Z 712.036,A -85,B 0,C 180,E1 -3544.603,E2 -3544.603} C_VEL
LIN {X 0,Y 520.667,Z 701.897,A -85,B 0,C 180,E1 -3546.053,E2 -3546.053} C_VEL
LIN {X 0,Y 521.073,Z 689.476,A -85,B 0,C 180,E1 -3547.463,E2 -3547.463} C_VEL
LIN {X 0,Y 521.491,Z 676.573,A -85,B 0,C 180,E1 -3548.623,E2 -3548.623} C_VEL
LIN {X 0,Y 521.942,Z 662.32,A -85,B 0,C 180,E1 -3549.637,E2 -3549.637} C_VEL
LIN {X 0,Y 522.345,Z 648.167,A -85,B 0,C 180,E1 -3550.412,E2 -3550.412} C_VEL
LIN {X 0,Y 522.701,Z 631.66,A -85,B 0,C 180,E1 -3551.076,E2 -3551.076} C_VEL
LIN {X 0,Y 522.914,Z 615.706,A -85,B 0,C 180,E1 -3551.495,E2 -3551.495} C_VEL
LIN {X 0,Y 523.514,Z 479.738,A -85,B 0,C 180,E1 -3553.422,E2 -3553.422} C_VEL
LIN {X 0,Y 522.734,Z 473.073,A -85,B 0,C 180,E1 -3553.576,E2 -3553.576} C_VEL
LIN {X 0,Y 523.654,Z 429.594,A -85,B 0,C 180,E1 -3557.026,E2 -3557.026} C_VEL
LIN {X 0,Y 524.395,Z 391.914,A -85,B 0,C 180,E1 -3560.017,E2 -3560.017} C_VEL
LIN {X 0,Y 525.069,Z 354.99,A -85,B 0,C 180,E1 -3562.925,E2 -3562.925} C_VEL
LIN {X 0,Y 525.468,Z 315.98,A -85,B 0,C 180,E1 -3565.984,E2 -3565.984} C_VEL
LIN {X 0,Y 525.494,Z 287.797,A -85,B 0,C 180,E1 -3568.193,E2 -3568.193} C_VEL
LIN {X 0,Y 520.607,Z 272.052,A -85,B 0,C 180,E1 -3569.725,E2 -3569.725} C_VEL
LIN {X 0,Y 520.567,Z 271.642,A -85,B 0,C 180,E1 -3570.04,E2 -3570.04} C_VEL
LIN {X 0,Y 520.543,Z 271.643,A -85,B 0,C 180,E1 -3573.413,E2 -3573.413} C_VEL
LIN {X 0,Y 520.579,Z 271.64,A -85,B 0,C 180,E1 -3576.812,E2 -3576.812} C_VEL
LIN {X 0,Y 520.578,Z 271.644,A -85,B 0,C 180,E1 -3580.242,E2 -3580.242} C_VEL
LIN {X 0,Y 520.542,Z 271.642,A -85,B 0,C 180,E1 -3583.599,E2 -3583.599} C_VEL
LIN {X 0,Y 520.57,Z 271.638,A -85,B 0,C 180,E1 -3587.013,E2 -3587.013} C_VEL
LIN {X 0,Y 520.587,Z 271.641,A -85,B 0,C 180,E1 -3590.492,E2 -3590.492} C_VEL
LIN {X 0,Y 520.546,Z 271.64,A -85,B 0,C 180,E1 -3593.825,E2 -3593.825} C_VEL
LIN {X 0,Y 520.561,Z 271.638,A -85,B 0,C 180,E1 -3597.247,E2 -3597.247} C_VEL
LIN {X 0,Y 520.59,Z 271.638,A -85,B 0,C 180,E1 -3600.66,E2 -3600.66} C_VEL
LIN {X 0,Y 520.554,Z 271.64,A -85,B 0,C 180,E1 -3604.075,E2 -3604.075} C_VEL
LIN {X 0,Y 520.552,Z 271.638,A -85,B 0,C 180,E1 -3607.616,E2 -3607.616} C_VEL
LIN {X 0,Y 520.587,Z 271.637,A -85,B 0,C 180,E1 -3610.961,E2 -3610.961} C_VEL
LIN {X 0,Y 520.574,Z 271.642,A -85,B 0,C 180,E1 -3614.459,E2 -3614.459} C_VEL
LIN {X 0,Y 520.549,Z 271.639,A -85,B 0,C 180,E1 -3617.898,E2 -3617.898} C_VEL
LIN {X 0,Y 520.578,Z 271.634,A -85,B 0,C 180,E1 -3621.331,E2 -3621.331} C_VEL
LIN {X 0,Y 520.587,Z 271.64,A -85,B 0,C 180,E1 -3624.752,E2 -3624.752} C_VEL
LIN {X 0,Y 520.554,Z 271.64,A -85,B 0,C 180,E1 -3628.197,E2 -3628.197} C_VEL
LIN {X 0,Y 520.558,Z 271.637,A -85,B 0,C 180,E1 -3631.754,E2 -3631.754} C_VEL
LIN {X 0,Y 520.587,Z 271.637,A -85,B 0,C 180,E1 -3635.183,E2 -3635.183} C_VEL
LIN {X 0,Y 520.573,Z 271.642,A -85,B 0,C 180,E1 -3638.625,E2 -3638.625} C_VEL
LIN {X 0,Y 520.554,Z 271.64,A -85,B 0,C 180,E1 -3642.093,E2 -3642.093} C_VEL
LIN {X 0,Y 520.584,Z 271.637,A -85,B 0,C 180,E1 -3645.492,E2 -3645.492} C_VEL
LIN {X 0,Y 520.589,Z 271.641,A -85,B 0,C 180,E1 -3649.008,E2 -3649.008} C_VEL
LIN {X 0,Y 520.553,Z 271.631,A -85,B 0,C 180,E1 -3652.355,E2 -3652.355} C_VEL
LIN {X 0,Y 520.609,Z 271.883,A -85,B 0,C 180,E1 -3653.768,E2 -3653.768} C_VEL
LIN {X 0,Y 522.835,Z 277.781,A -85,B 0,C 180,E1 -3654.456,E2 -3654.456} C_VEL
LIN {X 0,Y 529.438,Z 295.079,A -85,B 0,C 180,E1 -3656.276,E2 -3656.276} C_VEL
LIN {X 0,Y 528.74,Z 316.137,A -85,B 0,C 180,E1 -3657.792,E2 -3657.792} C_VEL
LIN {X 0,Y 530.995,Z 330.738,A -85,B 0,C 180,E1 -3658.163,E2 -3658.163} C_VEL
LIN {X 0,Y 529.192,Z 533.372,A -85,B 0,C 180,E1 -3661.125,E2 -3661.125} C_VEL
LIN {X 0,Y 528.748,Z 578.449,A -85,B 0,C 180,E1 -3661.804,E2 -3661.804} C_VEL
LIN {X 0,Y 528.168,Z 599.563,A -85,B 0,C 180,E1 -3662.331,E2 -3662.331} C_VEL
LIN {X 0,Y 527.46,Z 619.053,A -85,B 0,C 180,E1 -3663.021,E2 -3663.021} C_VEL
LIN {X 0,Y 526.617,Z 638.315,A -85,B 0,C 180,E1 -3663.904,E2 -3663.904} C_VEL
LIN {X 0,Y 525.65,Z 657.848,A -85,B 0,C 180,E1 -3665.023,E2 -3665.023} C_VEL
LIN {X 0,Y 524.688,Z 675.99,A -85,B 0,C 180,E1 -3666.293,E2 -3666.293} C_VEL
LIN {X 0,Y 523.735,Z 693.189,A -85,B 0,C 180,E1 -3667.733,E2 -3667.733} C_VEL
LIN {X 0,Y 522.831,Z 709.385,A -85,B 0,C 180,E1 -3669.341,E2 -3669.341} C_VEL
LIN {X 0,Y 522.006,Z 724.518,A -85,B 0,C 180,E1 -3671.122,E2 -3671.122} C_VEL
LIN {X 0,Y 521.321,Z 738.359,A -85,B 0,C 180,E1 -3673.052,E2 -3673.052} C_VEL
LIN {X 0,Y 520.808,Z 750.021,A -85,B 0,C 180,E1 -3674.98,E2 -3674.98} C_VEL
LIN {X 0,Y 520.406,Z 760.854,A -85,B 0,C 180,E1 -3677.124,E2 -3677.124} C_VEL
LIN {X 0,Y 520.153,Z 770.066,A -85,B 0,C 180,E1 -3679.367,E2 -3679.367} C_VEL
LIN {X 0,Y 520.012,Z 777.295,A -85,B 0,C 180,E1 -3681.599,E2 -3681.599} C_VEL
LIN {X 0,Y 519.946,Z 782.733,A -85,B 0,C 180,E1 -3683.821,E2 -3683.821} C_VEL
LIN {X 0,Y 519.919,Z 786.405,A -85,B 0,C 180,E1 -3686.031,E2 -3686.031} C_VEL
LIN {X 0,Y 519.907,Z 788.443,A -85,B 0,C 180,E1 -3688.238,E2 -3688.238} C_VEL
LIN {X 0,Y 519.9,Z 788.895,A -85,B 0,C 180,E1 -3690.552,E2 -3690.552} C_VEL
LIN {X 0,Y 519.911,Z 787.729,A -85,B 0,C 180,E1 -3692.757,E2 -3692.757} C_VEL
LIN {X 0,Y 519.92,Z 784.881,A -85,B 0,C 180,E1 -3695.021,E2 -3695.021} C_VEL
LIN {X 0,Y 519.953,Z 780.479,A -85,B 0,C 180,E1 -3697.182,E2 -3697.182} C_VEL
LIN {X 0,Y 520.044,Z 774.616,A -85,B 0,C 180,E1 -3699.295,E2 -3699.295} C_VEL
LIN {X 0,Y 520.225,Z 767.086,A -85,B 0,C 180,E1 -3701.42,E2 -3701.42} C_VEL
LIN {X 0,Y 520.523,Z 757.703,A -85,B 0,C 180,E1 -3703.554,E2 -3703.554} C_VEL
LIN {X 0,Y 520.943,Z 746.823,A -85,B 0,C 180,E1 -3705.588,E2 -3705.588} C_VEL
LIN {X 0,Y 521.506,Z 734.493,A -85,B 0,C 180,E1 -3707.519,E2 -3707.519} C_VEL
LIN {X 0,Y 522.2,Z 720.731,A -85,B 0,C 180,E1 -3709.345,E2 -3709.345} C_VEL
LIN {X 0,Y 523.025,Z 705.489,A -85,B 0,C 180,E1 -3711.064,E2 -3711.064} C_VEL
LIN {X 0,Y 523.971,Z 688.603,A -85,B 0,C 180,E1 -3712.673,E2 -3712.673} C_VEL
LIN {X 0,Y 524.948,Z 671.36,A -85,B 0,C 180,E1 -3714.055,E2 -3714.055} C_VEL
LIN {X 0,Y 525.91,Z 653.42,A -85,B 0,C 180,E1 -3715.257,E2 -3715.257} C_VEL
LIN {X 0,Y 526.807,Z 634.182,A -85,B 0,C 180,E1 -3716.307,E2 -3716.307} C_VEL
LIN {X 0,Y 527.624,Z 614.8,A -85,B 0,C 180,E1 -3717.145,E2 -3717.145} C_VEL
LIN {X 0,Y 528.309,Z 594.391,A -85,B 0,C 180,E1 -3717.813,E2 -3717.813} C_VEL
LIN {X 0,Y 528.817,Z 573.178,A -85,B 0,C 180,E1 -3718.29,E2 -3718.29} C_VEL
LIN {X 0,Y 530.518,Z 341.093,A -85,B 0,C 180,E1 -3721.606,E2 -3721.606} C_VEL
LIN {X 0,Y 530.379,Z 327.998,A -85,B 0,C 180,E1 -3721.81,E2 -3721.81} C_VEL
LIN {X 0,Y 528.39,Z 316.056,A -85,B 0,C 180,E1 -3722.123,E2 -3722.123} C_VEL
LIN {X 0,Y 528.883,Z 294.028,A -85,B 0,C 180,E1 -3723.714,E2 -3723.714} C_VEL
LIN {X 0,Y 521.663,Z 274.863,A -85,B 0,C 180,E1 -3725.737,E2 -3725.737} C_VEL
LIN {X 0,Y 520.597,Z 271.853,A -85,B 0,C 180,E1 -3726.131,E2 -3726.131} C_VEL
LIN {X 0,Y 520.551,Z 271.644,A -85,B 0,C 180,E1 -3729.626,E2 -3729.626} C_VEL
LIN {X 0,Y 520.584,Z 271.642,A -85,B 0,C 180,E1 -3732.988,E2 -3732.988} C_VEL
LIN {X 0,Y 520.575,Z 271.641,A -85,B 0,C 180,E1 -3736.408,E2 -3736.408} C_VEL
LIN {X 0,Y 520.543,Z 271.645,A -85,B 0,C 180,E1 -3739.806,E2 -3739.806} C_VEL
LIN {X 0,Y 520.569,Z 271.644,A -85,B 0,C 180,E1 -3743.22,E2 -3743.22} C_VEL
LIN {X 0,Y 520.577,Z 271.875,A -85,B 0,C 180,E1 -3746.102,E2 -3746.102} C_VEL
LIN {X 0,Y 524.315,Z 282.062,A -85,B 0,C 180,E1 -3747.447,E2 -3747.447} C_VEL
LIN {X 0,Y 527.874,Z 293.038,A -85,B 0,C 180,E1 -3748.736,E2 -3748.736} C_VEL
LIN {X 0,Y 525.988,Z 334.41,A -85,B 0,C 180,E1 -3752.305,E2 -3752.305} C_VEL
LIN {X 0,Y 525.771,Z 342.541,A -85,B 0,C 180,E1 -3752.955,E2 -3752.955} C_VEL
LIN {X 0,Y 527.928,Z 356.398,A -85,B 0,C 180,E1 -3753.293,E2 -3753.293} C_VEL
LIN {X 0,Y 526.234,Z 559.761,A -85,B 0,C 180,E1 -3756.239,E2 -3756.239} C_VEL
LIN {X 0,Y 525.776,Z 579.393,A -85,B 0,C 180,E1 -3756.73,E2 -3756.73} C_VEL
LIN {X 0,Y 525.193,Z 598.474,A -85,B 0,C 180,E1 -3757.421,E2 -3757.421} C_VEL
LIN {X 0,Y 524.498,Z 616.529,A -85,B 0,C 180,E1 -3758.296,E2 -3758.296} C_VEL
LIN {X 0,Y 523.739,Z 634.212,A -85,B 0,C 180,E1 -3759.377,E2 -3759.377} C_VEL
LIN {X 0,Y 523.02,Z 650.143,A -85,B 0,C 180,E1 -3760.571,E2 -3760.571} C_VEL
LIN {X 0,Y 522.275,Z 665.726,A -85,B 0,C 180,E1 -3761.99,E2 -3761.99} C_VEL
LIN {X 0,Y 521.623,Z 679.741,A -85,B 0,C 180,E1 -3763.52,E2 -3763.52} C_VEL
LIN {X 0,Y 521.059,Z 692.752,A -85,B 0,C 180,E1 -3765.214,E2 -3765.214} C_VEL
LIN {X 0,Y 520.616,Z 704.206,A -85,B 0,C 180,E1 -3767.015,E2 -3767.015} C_VEL
LIN {X 0,Y 520.299,Z 714.139,A -85,B 0,C 180,E1 -3768.921,E2 -3768.921} C_VEL
LIN {X 0,Y 520.094,Z 722.571,A -85,B 0,C 180,E1 -3770.93,E2 -3770.93} C_VEL
LIN {X 0,Y 519.98,Z 729.129,A -85,B 0,C 180,E1 -3772.931,E2 -3772.931} C_VEL
LIN {X 0,Y 519.934,Z 734.156,A -85,B 0,C 180,E1 -3775.036,E2 -3775.036} C_VEL
LIN {X 0,Y 519.913,Z 737.337,A -85,B 0,C 180,E1 -3777.134,E2 -3777.134} C_VEL
LIN {X 0,Y 519.917,Z 738.829,A -85,B 0,C 180,E1 -3779.229,E2 -3779.229} C_VEL
LIN {X 0,Y 519.911,Z 738.672,A -85,B 0,C 180,E1 -3781.323,E2 -3781.323} C_VEL
LIN {X 0,Y 519.914,Z 736.798,A -85,B 0,C 180,E1 -3783.418,E2 -3783.418} C_VEL
LIN {X 0,Y 519.936,Z 733.173,A -85,B 0,C 180,E1 -3785.518,E2 -3785.518} C_VEL
LIN {X 0,Y 519.996,Z 727.749,A -85,B 0,C 180,E1 -3787.625,E2 -3787.625} C_VEL
LIN {X 0,Y 520.14,Z 720.827,A -85,B 0,C 180,E1 -3789.628,E2 -3789.628} C_VEL
LIN {X 0,Y 520.373,Z 711.91,A -85,B 0,C 180,E1 -3791.64,E2 -3791.64} C_VEL
LIN {X 0,Y 520.72,Z 701.384,A -85,B 0,C 180,E1 -3793.548,E2 -3793.548} C_VEL
LIN {X 0,Y 521.195,Z 689.297,A -85,B 0,C 180,E1 -3795.352,E2 -3795.352} C_VEL
LIN {X 0,Y 521.799,Z 675.599,A -85,B 0,C 180,E1 -3797.049,E2 -3797.049} C_VEL
LIN {X 0,Y 522.47,Z 661.351,A -85,B 0,C 180,E1 -3798.523,E2 -3798.523} C_VEL
LIN {X 0,Y 523.246,Z 645.093,A -85,B 0,C 180,E1 -3799.922,E2 -3799.922} C_VEL
LIN {X 0,Y 523.989,Z 628.721,A -85,B 0,C 180,E1 -3801.077,E2 -3801.077} C_VEL
LIN {X 0,Y 524.744,Z 610.55,A -85,B 0,C 180,E1 -3802.106,E2 -3802.106} C_VEL
LIN {X 0,Y 525.405,Z 592.299,A -85,B 0,C 180,E1 -3802.917,E2 -3802.917} C_VEL
LIN {X 0,Y 525.935,Z 573.232,A -85,B 0,C 180,E1 -3803.539,E2 -3803.539} C_VEL
LIN {X 0,Y 526.317,Z 553.452,A -85,B 0,C 180,E1 -3803.961,E2 -3803.961} C_VEL
LIN {X 0,Y 527.04,Z 459.968,A -85,B 0,C 180,E1 -3805.307,E2 -3805.307} C_VEL
LIN {X 0,Y 526.195,Z 452.38,A -85,B 0,C 180,E1 -3805.463,E2 -3805.463} C_VEL
LIN {X 0,Y 520.736,Z 432.549,A -85,B 0,C 180,E1 -3806.046,E2 -3806.046} C_VEL
LIN {X 0,Y 520.123,Z 426.027,A -85,B 0,C 180,E1 -3806.177,E2 -3806.177} C_VEL
LIN {X 0,Y 520.602,Z 355.073,A -85,B 0,C 180,E1 -3807.23,E2 -3807.23} C_VEL
LIN {X 0,Y 518.426,Z 341.796,A -85,B 0,C 180,E1 -3807.604,E2 -3807.604} C_VEL
LIN {X 0,Y 520.253,Z 299.007,A -85,B 0,C 180,E1 -3811.259,E2 -3811.259} C_VEL
LIN {X 0,Y 520.238,Z 294.715,A -85,B 0,C 180,E1 -3811.648,E2 -3811.648} C_VEL
LIN {X 0,Y 513.404,Z 275.245,A -85,B 0,C 180,E1 -3813.937,E2 -3813.937} C_VEL
LIN {X 0,Y 512.629,Z 272.811,A -85,B 0,C 180,E1 -3814.277,E2 -3814.277} C_VEL
LIN {X 0,Y 512.641,Z 272.625,A -85,B 0,C 180,E1 -3817.484,E2 -3817.484} C_VEL
LIN {X 0,Y 512.649,Z 272.627,A -85,B 0,C 180,E1 -3820.991,E2 -3820.991} C_VEL
LIN {X 0,Y 512.631,Z 272.627,A -85,B 0,C 180,E1 -3824.449,E2 -3824.449} C_VEL
LIN {X 0,Y 512.63,Z 272.628,A -85,B 0,C 180,E1 -3828.009,E2 -3828.009} C_VEL
LIN {X 0,Y 512.649,Z 272.624,A -85,B 0,C 180,E1 -3831.524,E2 -3831.524} C_VEL
LIN {X 0,Y 512.631,Z 272.628,A -85,B 0,C 180,E1 -3835.009,E2 -3835.009} C_VEL
LIN {X 0,Y 512.644,Z 272.63,A -85,B 0,C 180,E1 -3838.485,E2 -3838.485} C_VEL
LIN {X 0,Y 512.648,Z 272.623,A -85,B 0,C 180,E1 -3841.962,E2 -3841.962} C_VEL
LIN {X 0,Y 512.627,Z 272.62,A -85,B 0,C 180,E1 -3845.451,E2 -3845.451} C_VEL
LIN {X 0,Y 512.605,Z 272.627,A -85,B 0,C 180,E1 -3848.847,E2 -3848.847} C_VEL
LIN {X 0,Y 512.64,Z 272.625,A -85,B 0,C 180,E1 -3852.168,E2 -3852.168} C_VEL
LIN {X 0,Y 512.61,Z 272.609,A -85,B 0,C 180,E1 -3855.541,E2 -3855.541} C_VEL
LIN {X 0,Y 512.577,Z 272.624,A -85,B 0,C 180,E1 -3858.869,E2 -3858.869} C_VEL
LIN {X 0,Y 512.662,Z 272.926,A -85,B 0,C 180,E1 -3859.691,E2 -3859.691} C_VEL
LIN {X 0,Y 518.697,Z 292.075,A -85,B 0,C 180,E1 -3861.658,E2 -3861.658} C_VEL
LIN {X 0,Y 518.15,Z 331.621,A -85,B 0,C 180,E1 -3864.851,E2 -3864.851} C_VEL
LIN {X 0,Y 517.386,Z 372.895,A -85,B 0,C 180,E1 -3868.172,E2 -3868.172} C_VEL
LIN {X 0,Y 516.402,Z 417.038,A -85,B 0,C 180,E1 -3871.719,E2 -3871.719} C_VEL
LIN {X 0,Y 515.379,Z 461.419,A -85,B 0,C 180,E1 -3875.286,E2 -3875.286} C_VEL
LIN {X 0,Y 515.161,Z 474.189,A -85,B 0,C 180,E1 -3876.273,E2 -3876.273} C_VEL
LIN {X 0,Y 516.114,Z 484.411,A -85,B 0,C 180,E1 -3876.461,E2 -3876.461} C_VEL
LIN {X 0,Y 515.251,Z 616.503,A -85,B 0,C 180,E1 -3878.357,E2 -3878.357} C_VEL
LIN {X 0,Y 515.005,Z 632.345,A -85,B 0,C 180,E1 -3878.785,E2 -3878.785} C_VEL
LIN {X 0,Y 514.623,Z 648.552,A -85,B 0,C 180,E1 -3879.448,E2 -3879.448} C_VEL
LIN {X 0,Y 514.176,Z 663.264,A -85,B 0,C 180,E1 -3880.272,E2 -3880.272} C_VEL
LIN {X 0,Y 513.662,Z 677.86,A -85,B 0,C 180,E1 -3881.337,E2 -3881.337} C_VEL
LIN {X 0,Y 513.218,Z 690.291,A -85,B 0,C 180,E1 -3882.488,E2 -3882.488} C_VEL
LIN {X 0,Y 512.785,Z 702.303,A -85,B 0,C 180,E1 -3883.875,E2 -3883.875} C_VEL
LIN {X 0,Y 512.461,Z 711.979,A -85,B 0,C 180,E1 -3885.27,E2 -3885.27} C_VEL
LIN {X 0,Y 512.198,Z 721.204,A -85,B 0,C 180,E1 -3886.954,E2 -3886.954} C_VEL
LIN {X 0,Y 512.048,Z 727.969,A -85,B 0,C 180,E1 -3888.558,E2 -3888.558} C_VEL
LIN {X 0,Y 511.963,Z 733.565,A -85,B 0,C 180,E1 -3890.373,E2 -3890.373} C_VEL
LIN {X 0,Y 511.936,Z 737.182,A -85,B 0,C 180,E1 -3892.143,E2 -3892.143} C_VEL
LIN {X 0,Y 511.927,Z 739.08,A -85,B 0,C 180,E1 -3893.968,E2 -3893.968} C_VEL
LIN {X 0,Y 511.926,Z 739.258,A -85,B 0,C 180,E1 -3895.818,E2 -3895.818} C_VEL
LIN {X 0,Y 511.931,Z 737.529,A -85,B 0,C 180,E1 -3897.698,E2 -3897.698} C_VEL
LIN {X 0,Y 511.959,Z 734.186,A -85,B 0,C 180,E1 -3899.481,E2 -3899.481} C_VEL
LIN {X 0,Y 512.028,Z 729.131,A -85,B 0,C 180,E1 -3901.206,E2 -3901.206} C_VEL
LIN {X 0,Y 512.176,Z 722.266,A -85,B 0,C 180,E1 -3902.918,E2 -3902.918} C_VEL
LIN {X 0,Y 512.399,Z 714.171,A -85,B 0,C 180,E1 -3904.462,E2 -3904.462} C_VEL
LIN {X 0,Y 512.724,Z 704.172,A -85,B 0,C 180,E1 -3905.973,E2 -3905.973} C_VEL
LIN {X 0,Y 513.121,Z 693.219,A -85,B 0,C 180,E1 -3907.299,E2 -3907.299} C_VEL
LIN {X 0,Y 513.602,Z 679.796,A -85,B 0,C 180,E1 -3908.595,E2 -3908.595} C_VEL
LIN {X 0,Y 514.085,Z 666.102,A -85,B 0,C 180,E1 -3909.636,E2 -3909.636} C_VEL
LIN {X 0,Y 514.554,Z 651.211,A -85,B 0,C 180,E1 -3910.513,E2 -3910.513} C_VEL
LIN {X 0,Y 514.943,Z 635.865,A -85,B 0,C 180,E1 -3911.183,E2 -3911.183} C_VEL
LIN {X 0,Y 515.215,Z 619.068,A -85,B 0,C 180,E1 -3911.68,E2 -3911.68} C_VEL
LIN {X 0,Y 515.387,Z 595.185,A -85,B 0,C 180,E1 -3912.064,E2 -3912.064} C_VEL
LIN {X 0,Y 515.916,Z 480.468,A -85,B 0,C 180,E1 -3913.695,E2 -3913.695} C_VEL
LIN {X 0,Y 515.086,Z 473.319,A -85,B 0,C 180,E1 -3913.865,E2 -3913.865} C_VEL
LIN {X 0,Y 516.078,Z 429.056,A -85,B 0,C 180,E1 -3917.408,E2 -3917.408} C_VEL
LIN {X 0,Y 516.988,Z 388.843,A -85,B 0,C 180,E1 -3920.627,E2 -3920.627} C_VEL
LIN {X 0,Y 517.686,Z 347.255,A -85,B 0,C 180,E1 -3923.908,E2 -3923.908} C_VEL
LIN {X 0,Y 518.126,Z 307.146,A -85,B 0,C 180,E1 -3927.078,E2 -3927.078} C_VEL
LIN {X 0,Y 518.1,Z 290.356,A -85,B 0,C 180,E1 -3928.401,E2 -3928.401} C_VEL
LIN {X 0,Y 512.693,Z 273.013,A -85,B 0,C 180,E1 -3930.113,E2 -3930.113} C_VEL
LIN {X 0,Y 512.654,Z 272.631,A -85,B 0,C 180,E1 -3930.438,E2 -3930.438} C_VEL
LIN {X 0,Y 512.614,Z 272.635,A -85,B 0,C 180,E1 -3933.844,E2 -3933.844} C_VEL
LIN {X 0,Y 512.607,Z 272.631,A -85,B 0,C 180,E1 -3937.305,E2 -3937.305} C_VEL
LIN {X 0,Y 512.645,Z 272.624,A -85,B 0,C 180,E1 -3940.754,E2 -3940.754} C_VEL
LIN {X 0,Y 512.639,Z 272.627,A -85,B 0,C 180,E1 -3944.269,E2 -3944.269} C_VEL
LIN {X 0,Y 512.606,Z 272.63,A -85,B 0,C 180,E1 -3947.724,E2 -3947.724} C_VEL
LIN {X 0,Y 512.619,Z 272.626,A -85,B 0,C 180,E1 -3951.249,E2 -3951.249} C_VEL
LIN {X 0,Y 512.649,Z 272.629,A -85,B 0,C 180,E1 -3954.628,E2 -3954.628} C_VEL
LIN {X 0,Y 512.618,Z 272.631,A -85,B 0,C 180,E1 -3958.099,E2 -3958.099} C_VEL
LIN {X 0,Y 512.61,Z 272.626,A -85,B 0,C 180,E1 -3961.564,E2 -3961.564} C_VEL
LIN {X 0,Y 512.644,Z 272.626,A -85,B 0,C 180,E1 -3965.035,E2 -3965.035} C_VEL
LIN {X 0,Y 512.646,Z 272.63,A -85,B 0,C 180,E1 -3968.579,E2 -3968.579} C_VEL
LIN {X 0,Y 512.613,Z 272.629,A -85,B 0,C 180,E1 -3972.046,E2 -3972.046} C_VEL
LIN {X 0,Y 512.615,Z 272.625,A -85,B 0,C 180,E1 -3975.615,E2 -3975.615} C_VEL
LIN {X 0,Y 512.649,Z 272.626,A -85,B 0,C 180,E1 -3979.008,E2 -3979.008} C_VEL
LIN {X 0,Y 512.633,Z 272.629,A -85,B 0,C 180,E1 -3982.475,E2 -3982.475} C_VEL
LIN {X 0,Y 512.612,Z 272.628,A -85,B 0,C 180,E1 -3985.953,E2 -3985.953} C_VEL
LIN {X 0,Y 512.639,Z 272.623,A -85,B 0,C 180,E1 -3989.439,E2 -3989.439} C_VEL
LIN {X 0,Y 512.649,Z 272.629,A -85,B 0,C 180,E1 -3992.967,E2 -3992.967} C_VEL
LIN {X 0,Y 512.619,Z 272.63,A -85,B 0,C 180,E1 -3996.366,E2 -3996.366} C_VEL
LIN {X 0,Y 512.619,Z 272.627,A -85,B 0,C 180,E1 -3999.919,E2 -3999.919} C_VEL
LIN {X 0,Y 512.648,Z 272.628,A -85,B 0,C 180,E1 -4003.356,E2 -4003.356} C_VEL
LIN {X 0,Y 512.643,Z 272.631,A -85,B 0,C 180,E1 -4006.84,E2 -4006.84} C_VEL
LIN {X 0,Y 512.615,Z 272.631,A -85,B 0,C 180,E1 -4010.228,E2 -4010.228} C_VEL
LIN {X 0,Y 512.681,Z 272.863,A -85,B 0,C 180,E1 -4013.217,E2 -4013.217} C_VEL
LIN {X 0,Y 514.781,Z 278.552,A -85,B 0,C 180,E1 -4013.9,E2 -4013.9} C_VEL
LIN {X 0,Y 522.312,Z 298.215,A -85,B 0,C 180,E1 -4016.017,E2 -4016.017} C_VEL
LIN {X 0,Y 521.644,Z 316.225,A -85,B 0,C 180,E1 -4017.331,E2 -4017.331} C_VEL
LIN {X 0,Y 524.062,Z 331.98,A -85,B 0,C 180,E1 -4017.743,E2 -4017.743} C_VEL
LIN {X 0,Y 522.004,Z 524.959,A -85,B 0,C 180,E1 -4020.635,E2 -4020.635} C_VEL
LIN {X 0,Y 521.467,Z 578.492,A -85,B 0,C 180,E1 -4021.44,E2 -4021.44} C_VEL
LIN {X 0,Y 520.875,Z 600.034,A -85,B 0,C 180,E1 -4021.974,E2 -4021.974} C_VEL
LIN {X 0,Y 520.123,Z 620.862,A -85,B 0,C 180,E1 -4022.713,E2 -4022.713} C_VEL
LIN {X 0,Y 519.281,Z 639.847,A -85,B 0,C 180,E1 -4023.592,E2 -4023.592} C_VEL
LIN {X 0,Y 518.247,Z 658.777,A -85,B 0,C 180,E1 -4024.705,E2 -4024.705} C_VEL
LIN {X 0,Y 517.144,Z 677.456,A -85,B 0,C 180,E1 -4026.047,E2 -4026.047} C_VEL
LIN {X 0,Y 516.143,Z 693.796,A -85,B 0,C 180,E1 -4027.447,E2 -4027.447} C_VEL
LIN {X 0,Y 515.145,Z 709.904,A -85,B 0,C 180,E1 -4029.078,E2 -4029.078} C_VEL
LIN {X 0,Y 514.219,Z 725.369,A -85,B 0,C 180,E1 -4030.935,E2 -4030.935} C_VEL
LIN {X 0,Y 513.443,Z 739.579,A -85,B 0,C 180,E1 -4032.97,E2 -4032.97} C_VEL
LIN {X 0,Y 512.849,Z 751.925,A -85,B 0,C 180,E1 -4035.089,E2 -4035.089} C_VEL
LIN {X 0,Y 512.439,Z 761.882,A -85,B 0,C 180,E1 -4037.149,E2 -4037.149} C_VEL
LIN {X 0,Y 512.173,Z 770.471,A -85,B 0,C 180,E1 -4039.314,E2 -4039.314} C_VEL
LIN {X 0,Y 512.019,Z 777.598,A -85,B 0,C 180,E1 -4041.58,E2 -4041.58} C_VEL
LIN {X 0,Y 511.948,Z 782.936,A -85,B 0,C 180,E1 -4043.835,E2 -4043.835} C_VEL
LIN {X 0,Y 511.918,Z 786.563,A -85,B 0,C 180,E1 -4046.081,E2 -4046.081} C_VEL
LIN {X 0,Y 511.904,Z 788.51,A -85,B 0,C 180,E1 -4048.322,E2 -4048.322} C_VEL
LIN {X 0,Y 511.9,Z 788.895,A -85,B 0,C 180,E1 -4050.561,E2 -4050.561} C_VEL
